C07281=1053.248,31.151,424.768,170.927,31.729,155.954
C07282=1053.242,30.901,424.785,170.926,31.727,155.954
C07283=1053.236,30.652,424.801,170.924,31.725,155.953
C07284=1053.230,30.403,424.817,170.922,31.723,155.953
C07285=1053.224,30.153,424.833,170.920,31.720,155.953
C07286=1053.217,29.868,424.851,170.919,31.718,155.952
C07287=1053.209,29.582,424.870,170.917,31.716,155.952
C07288=1053.203,29.296,424.888,170.915,31.714,155.952
C07289=1053.196,29.011,424.906,170.914,31.711,155.951
C07290=1053.189,28.761,424.923,170.912,31.709,155.951
C07291=1053.184,28.511,424.938,170.910,31.707,155.951
C07292=1053.177,28.262,424.954,170.909,31.704,155.950
C07293=1053.171,28.012,424.970,170.907,31.702,155.950
C07294=1053.165,27.763,424.987,170.905,31.700,155.950
C07295=1053.158,27.514,425.002,170.903,31.698,155.949
C07296=1053.153,27.264,425.018,170.902,31.696,155.949
C07297=1053.146,27.015,425.034,170.900,31.694,155.949
C07298=1053.140,26.765,425.050,170.899,31.692,155.949
C07299=1053.134,26.516,425.066,170.897,31.690,155.948
C07300=1053.127,26.267,425.082,170.896,31.688,155.948
C07301=1053.122,26.017,425.097,170.894,31.686,155.948
C07302=1053.114,25.767,425.113,170.892,31.684,155.947
C07303=1053.108,25.518,425.130,170.891,31.682,155.947
C07304=1053.103,25.269,425.146,170.889,31.679,155.947
C07305=1053.096,25.019,425.161,170.887,31.677,155.946
C07306=1053.090,24.770,425.177,170.885,31.675,155.946
C07307=1053.084,24.521,425.193,170.884,31.673,155.946
C07308=1053.078,24.271,425.208,170.883,31.671,155.945
C07309=1053.071,24.022,425.224,170.881,31.669,155.945
C07310=1053.065,23.772,425.240,170.880,31.667,155.945
C07311=1053.059,23.523,425.256,170.878,31.665,155.945
C07312=1053.053,23.273,425.271,170.876,31.663,155.944
C07313=1053.047,23.024,425.288,170.874,31.660,155.944
C07314=1053.040,22.775,425.303,170.873,31.659,155.944
C07315=1053.035,22.525,425.319,170.871,31.656,155.943
C07316=1053.028,22.276,425.334,170.869,31.654,155.943
C07317=1053.022,22.026,425.350,170.868,31.652,155.943
C07318=1053.016,21.777,425.366,170.867,31.650,155.942
C07319=1053.010,21.528,425.382,170.865,31.648,155.942
C07320=1053.003,21.278,425.397,170.863,31.645,155.942
C07321=1052.997,21.029,425.413,170.862,31.644,155.942
C07322=1052.991,20.779,425.429,170.860,31.641,155.941
C07323=1052.985,20.530,425.444,170.858,31.639,155.941
C07324=1052.979,20.280,425.461,170.856,31.637,155.941
C07325=1052.973,20.030,425.475,170.855,31.635,155.940
C07326=1052.967,19.781,425.492,170.853,31.633,155.940
C07327=1052.960,19.531,425.507,170.852,31.631,155.940
C07328=1052.954,19.282,425.522,170.850,31.629,155.939
C07329=1052.948,19.032,425.538,170.849,31.627,155.939
C07330=1052.941,18.783,425.554,170.847,31.625,155.939
C07331=1052.936,18.533,425.569,170.845,31.623,155.939
C07332=1052.929,18.284,425.585,170.843,31.621,155.938
C07333=1052.923,18.035,425.600,170.842,31.619,155.938
C07334=1052.917,17.785,425.616,170.840,31.617,155.938
C07335=1052.910,17.536,425.631,170.838,31.615,155.937
C07336=1052.905,17.287,425.647,170.837,31.613,155.937
C07337=1052.898,17.037,425.662,170.836,31.611,155.937
C07338=1052.892,16.788,425.677,170.834,31.608,155.936
C07339=1052.886,16.538,425.693,170.832,31.606,155.936
C07340=1052.879,16.289,425.709,170.830,31.604,155.936
C07341=1052.874,16.039,425.724,170.829,31.602,155.936
C07342=1052.867,15.790,425.740,170.827,31.600,155.935
C07343=1052.861,15.541,425.755,170.825,31.598,155.935
C07344=1052.855,15.291,425.770,170.823,31.596,155.935
C07345=1052.848,15.042,425.786,170.823,31.594,155.934
C07346=1052.842,14.792,425.801,170.821,31.592,155.934
C07347=1052.836,14.543,425.817,170.819,31.590,155.934
C07348=1052.830,14.294,425.832,170.817,31.588,155.934
C07349=1052.824,14.044,425.847,170.816,31.586,155.933
C07350=1052.816,13.760,425.865,170.814,31.584,155.933
C07351=1052.809,13.475,425.882,170.812,31.581,155.933
C07352=1052.802,13.191,425.900,170.810,31.579,155.932
C07353=1052.795,12.906,425.917,170.808,31.577,155.932
C07354=1052.789,12.656,425.932,170.807,31.575,155.932
C07355=1052.782,12.407,425.948,170.805,31.573,155.931
C07356=1052.776,12.158,425.963,170.803,31.571,155.931
C07357=1052.769,11.908,425.978,170.802,31.569,155.931
C07358=1052.764,11.658,425.993,170.800,31.566,155.931
C07359=1052.757,11.409,426.009,170.798,31.564,155.930
C07360=1052.751,11.160,426.023,170.796,31.563,155.930
C07361=1052.745,10.910,426.038,170.794,31.561,155.930
C07362=1052.738,10.661,426.054,170.793,31.559,155.929
C07363=1052.732,10.412,426.069,170.792,31.557,155.929
C07364=1052.725,10.162,426.084,170.790,31.555,155.929
C07365=1052.719,9.912,426.099,170.788,31.553,155.929
C07366=1052.713,9.662,426.114,170.787,31.551,155.928
C07367=1052.707,9.414,426.130,170.785,31.548,155.928
C07368=1052.701,9.164,426.145,170.783,31.547,155.928
C07369=1052.695,8.915,426.159,170.781,31.545,155.928
C07370=1052.688,8.665,426.174,170.779,31.543,155.927
C07371=1052.682,8.415,426.189,170.778,31.541,155.927
C07372=1052.675,8.166,426.205,170.777,31.539,155.927
C07373=1052.669,7.917,426.220,170.775,31.537,155.926
C07374=1052.664,7.668,426.235,170.773,31.534,155.926
C07375=1052.657,7.418,426.250,170.772,31.533,155.926
C07376=1052.651,7.168,426.265,170.770,31.531,155.926
C07377=1052.645,6.919,426.280,170.768,31.529,155.925
C07378=1052.638,6.669,426.295,170.766,31.527,155.925
C07379=1052.632,6.421,426.310,170.764,31.525,155.925
C07380=1052.626,6.171,426.325,170.763,31.523,155.924
C07381=1052.619,5.921,426.340,170.762,31.521,155.924
C07382=1052.613,5.672,426.355,170.760,31.519,155.924
C07383=1052.607,5.422,426.370,170.758,31.516,155.924
C07384=1052.602,5.173,426.385,170.757,31.515,155.923
C07385=1052.595,4.923,426.400,170.755,31.513,155.923
C07386=1052.589,4.673,426.415,170.753,31.511,155.923
C07387=1052.582,4.424,426.430,170.751,31.509,155.922
C07388=1052.577,4.175,426.445,170.749,31.507,155.922
C07389=1052.570,3.925,426.460,170.749,31.505,155.922
C07390=1052.564,3.675,426.475,170.747,31.503,155.922
C07391=1052.557,3.426,426.489,170.745,31.500,155.921
C07392=1052.552,3.177,426.504,170.743,31.499,155.921
C07393=1052.545,2.927,426.519,170.741,31.497,155.921
C07394=1052.539,2.678,426.534,170.740,31.495,155.921
C07395=1052.533,2.429,426.549,170.738,31.493,155.920
C07396=1052.527,2.179,426.563,170.736,31.491,155.920
C07397=1052.521,1.929,426.579,170.734,31.489,155.920
C07398=1052.515,1.679,426.594,170.733,31.487,155.919
C07399=1052.509,1.430,426.609,170.732,31.485,155.919
C07400=1052.503,1.181,426.623,170.730,31.483,155.919
C07401=1052.496,0.931,426.638,170.728,31.481,155.919
C07402=1052.490,0.682,426.653,170.726,31.479,155.918
C07403=1052.484,0.432,426.668,170.725,31.477,155.918
C07404=1052.478,0.183,426.683,170.723,31.475,155.918
C07405=1052.472,-0.066,426.697,170.721,31.473,155.917
C07406=1052.465,-0.316,426.712,170.719,31.471,155.917
C07407=1052.459,-0.566,426.727,170.718,31.469,155.917
C07408=1052.453,-0.814,426.742,170.717,31.467,155.917
C07409=1052.447,-1.065,426.756,170.715,31.465,155.916
C07410=1052.441,-1.314,426.771,170.713,31.463,155.916
C07411=1052.435,-1.563,426.786,170.711,31.461,155.916
C07412=1052.429,-1.813,426.801,170.709,31.459,155.916
C07413=1052.422,-2.063,426.816,170.708,31.457,155.915
C07414=1052.415,-2.345,426.832,170.705,31.454,155.915
C07415=1052.409,-2.628,426.848,170.704,31.452,155.915
C07416=1052.402,-2.910,426.865,170.702,31.450,155.914
C07417=1052.395,-3.193,426.882,170.700,31.447,155.914
C07418=1052.389,-3.442,426.897,170.699,31.446,155.914
C07419=1052.383,-3.692,426.911,170.697,31.444,155.914
C07420=1052.377,-3.941,426.926,170.695,31.442,155.913
C07421=1052.369,-4.191,426.940,170.693,31.440,155.913
C07422=1052.364,-4.440,426.955,170.691,31.438,155.913
C07423=1052.358,-4.690,426.969,170.690,31.436,155.912
C07424=1052.351,-4.940,426.984,170.689,31.435,155.912
C07425=1052.345,-5.188,426.998,170.687,31.433,155.912
C07426=1052.338,-5.438,427.013,170.685,31.431,155.912
C07427=1052.333,-5.688,427.027,170.683,31.429,155.912
C07428=1052.326,-5.937,427.042,170.681,31.427,155.911
C07429=1052.319,-6.187,427.056,170.679,31.425,155.911
C07430=1052.314,-6.436,427.070,170.678,31.423,155.911
C07431=1052.307,-6.686,427.085,170.676,31.421,155.911
C07432=1052.301,-6.935,427.100,170.675,31.419,155.910
C07433=1052.295,-7.185,427.113,170.673,31.417,155.910
C07434=1052.288,-7.434,427.128,170.671,31.416,155.910
C07435=1052.283,-7.683,427.143,170.669,31.414,155.909
C07436=1052.276,-7.933,427.156,170.667,31.411,155.909
C07437=1052.270,-8.183,427.171,170.666,31.410,155.909
C07438=1052.264,-8.432,427.186,170.664,31.408,155.909
C07439=1052.258,-8.682,427.200,170.662,31.406,155.908
C07440=1052.251,-8.931,427.214,170.660,31.404,155.908
C07441=1052.245,-9.181,427.228,170.659,31.402,155.908
C07442=1052.239,-9.431,427.243,170.657,31.400,155.908
C07443=1052.232,-9.679,427.257,170.656,31.399,155.907
C07444=1052.226,-9.930,427.271,170.654,31.397,155.907
C07445=1052.220,-10.179,427.286,170.652,31.395,155.907
C07446=1052.213,-10.429,427.300,170.650,31.393,155.907
C07447=1052.208,-10.678,427.314,170.648,31.391,155.906
C07448=1052.202,-10.928,427.328,170.646,31.389,155.906
C07449=1052.195,-11.176,427.342,170.645,31.387,155.906
C07450=1052.189,-11.427,427.357,170.644,31.385,155.906
C07451=1052.183,-11.676,427.371,170.642,31.384,155.906
C07452=1052.177,-11.926,427.385,170.640,31.382,155.905
C07453=1052.171,-12.175,427.399,170.638,31.380,155.905
C07454=1052.165,-12.425,427.414,170.636,31.378,155.905
C07455=1052.159,-12.674,427.428,170.634,31.376,155.905
C07456=1052.152,-12.924,427.442,170.633,31.374,155.904
C07457=1052.146,-13.173,427.456,170.631,31.372,155.904
C07458=1052.140,-13.423,427.471,170.630,31.370,155.904
C07459=1052.134,-13.672,427.485,170.628,31.368,155.903
C07460=1052.127,-13.922,427.499,170.626,31.367,155.903
C07461=1052.122,-14.171,427.513,170.624,31.365,155.903
C07462=1052.115,-14.421,427.527,170.622,31.362,155.903
C07463=1052.109,-14.670,427.542,170.621,31.361,155.903
C07464=1052.102,-14.920,427.555,170.619,31.359,155.902
C07465=1052.097,-15.169,427.569,170.617,31.358,155.902
C07466=1052.090,-15.419,427.584,170.616,31.355,155.902
C07467=1052.084,-15.668,427.597,170.614,31.354,155.902
C07468=1052.077,-15.918,427.612,170.612,31.352,155.901
C07469=1052.072,-16.167,427.626,170.610,31.350,155.901
C07470=1052.065,-16.417,427.639,170.608,31.348,155.901
C07471=1052.059,-16.666,427.654,170.606,31.347,155.901
C07472=1052.052,-16.916,427.667,170.605,31.345,155.900
C07473=1052.047,-17.166,427.681,170.603,31.343,155.900
C07474=1052.040,-17.415,427.696,170.602,31.341,155.900
C07475=1052.034,-17.665,427.709,170.600,31.340,155.900
C07476=1052.027,-17.915,427.723,170.598,31.337,155.900
C07477=1052.021,-18.164,427.736,170.596,31.336,155.899
C07478=1052.014,-18.445,427.752,170.594,31.334,155.899
C07479=1052.007,-18.725,427.769,170.592,31.332,155.899
C07480=1052.000,-19.007,427.784,170.590,31.330,155.898
C07481=1051.993,-19.288,427.800,170.588,31.327,155.898
C07482=1051.987,-19.537,427.813,170.586,31.326,155.898
C07483=1051.980,-19.787,427.827,170.585,31.324,155.898
C07484=1051.975,-20.036,427.841,170.583,31.322,155.898
C07485=1051.967,-20.286,427.855,170.581,31.320,155.897
C07486=1051.962,-20.535,427.869,170.579,31.319,155.897
C07487=1051.956,-20.785,427.882,170.577,31.317,155.897
C07488=1051.949,-21.035,427.896,170.575,31.315,155.897
C07489=1051.943,-21.284,427.910,170.574,31.314,155.896
C07490=1051.936,-21.534,427.924,170.572,31.312,155.896
C07491=1051.931,-21.783,427.938,170.571,31.310,155.896
C07492=1051.925,-22.032,427.951,170.569,31.308,155.896
C07493=1051.918,-22.282,427.965,170.567,31.306,155.896
C07494=1051.912,-22.532,427.979,170.565,31.304,155.895
C07495=1051.906,-22.781,427.992,170.563,31.303,155.895
C07496=1051.900,-23.031,428.007,170.561,31.301,155.895
C07497=1051.894,-23.280,428.020,170.559,31.299,155.895
C07498=1051.887,-23.529,428.034,170.557,31.297,155.894
C07499=1051.881,-23.780,428.048,170.557,31.296,155.894
C07500=1051.875,-24.029,428.061,170.555,31.293,155.894
C07501=1051.869,-24.278,428.074,170.553,31.292,155.894
C07502=1051.863,-24.528,428.089,170.551,31.290,155.894
C07503=1051.857,-24.778,428.102,170.549,31.288,155.893
C07504=1051.850,-25.027,428.115,170.547,31.287,155.893
C07505=1051.844,-25.277,428.129,170.545,31.285,155.893
C07506=1051.838,-25.526,428.143,170.543,31.283,155.893
C07507=1051.832,-25.775,428.157,170.542,31.281,155.892
C07508=1051.825,-26.025,428.171,170.540,31.280,155.892
C07509=1051.819,-26.275,428.184,170.538,31.277,155.892
C07510=1051.814,-26.524,428.198,170.537,31.276,155.892
C07511=1051.807,-26.774,428.212,170.535,31.275,155.892
C07512=1051.801,-27.024,428.225,170.533,31.272,155.891
C07513=1051.795,-27.273,428.238,170.531,31.271,155.891
C07514=1051.788,-27.523,428.252,170.529,31.269,155.891
C07515=1051.782,-27.772,428.266,170.527,31.267,155.891
C07516=1051.776,-28.022,428.279,170.526,31.266,155.891
C07517=1051.769,-28.272,428.293,170.524,31.264,155.890
C07518=1051.763,-28.521,428.305,170.522,31.262,155.890
C07519=1051.757,-28.771,428.318,170.520,31.261,155.890
C07520=1051.751,-29.020,428.332,170.518,31.259,155.890
C07521=1051.744,-29.270,428.345,170.516,31.258,155.890
C07522=1051.739,-29.520,428.359,170.514,31.255,155.889
C07523=1051.732,-29.769,428.372,170.512,31.254,155.889
C07524=1051.726,-30.019,428.386,170.511,31.252,155.889
C07525=1051.719,-30.268,428.399,170.510,31.250,155.889
C07526=1051.713,-30.517,428.413,170.508,31.249,155.888
C07527=1051.707,-30.767,428.426,170.506,31.247,155.888
C07528=1051.700,-31.017,428.439,170.504,31.246,155.888
C07529=1051.694,-31.266,428.452,170.502,31.244,155.888
C07530=1051.688,-31.516,428.465,170.500,31.242,155.888
C07531=1051.682,-31.765,428.479,170.498,31.241,155.888
C07532=1051.676,-32.015,428.493,170.496,31.239,155.887
C07533=1051.669,-32.264,428.506,170.495,31.237,155.887
C07534=1051.664,-32.514,428.519,170.493,31.236,155.887
C07535=1051.657,-32.764,428.532,170.491,31.234,155.887
C07536=1051.651,-33.014,428.546,170.489,31.232,155.887
C07537=1051.644,-33.263,428.559,170.487,31.230,155.886
C07538=1051.638,-33.512,428.572,170.485,31.229,155.886
C07539=1051.632,-33.762,428.585,170.483,31.227,155.886
C07540=1051.626,-34.011,428.598,170.481,31.226,155.886
C07541=1051.619,-34.261,428.612,170.480,31.224,155.886
C07542=1051.613,-34.542,428.627,170.478,31.222,155.885
C07543=1051.606,-34.822,428.642,170.476,31.220,155.885
C07544=1051.599,-35.102,428.656,170.474,31.218,155.885
C07545=1051.592,-35.382,428.671,170.472,31.216,155.885
C07546=1051.586,-35.632,428.684,170.470,31.215,155.884
C07547=1051.580,-35.881,428.697,170.468,31.213,155.884
C07548=1051.573,-36.130,428.710,170.466,31.212,155.884
C07549=1051.567,-36.380,428.723,170.465,31.210,155.884
C07550=1051.561,-36.630,428.737,170.463,31.208,155.884
C07551=1051.554,-36.879,428.750,170.461,31.207,155.884
C07552=1051.548,-37.129,428.762,170.459,31.205,155.883
C07553=1051.542,-37.379,428.776,170.457,31.203,155.883
C07554=1051.537,-37.628,428.789,170.455,31.201,155.883
C07555=1051.531,-37.878,428.802,170.453,31.200,155.883
C07556=1051.525,-38.127,428.815,170.451,31.198,155.883
C07557=1051.518,-38.376,428.829,170.449,31.197,155.882
C07558=1051.512,-38.627,428.841,170.448,31.195,155.882
C07559=1051.506,-38.876,428.855,170.446,31.193,155.882
C07560=1051.499,-39.126,428.867,170.444,31.192,155.882
C07561=1051.493,-39.375,428.880,170.442,31.190,155.882
C07562=1051.487,-39.624,428.893,170.440,31.189,155.881
C07563=1051.481,-39.874,428.906,170.438,31.187,155.881
C07564=1051.475,-40.124,428.919,170.436,31.186,155.881
C07565=1051.468,-40.374,428.932,170.434,31.184,155.881
C07566=1051.461,-40.623,428.945,170.433,31.183,155.881
C07567=1051.455,-40.873,428.957,170.431,31.181,155.881
C07568=1051.449,-41.122,428.970,170.429,31.180,155.880
C07569=1051.443,-41.372,428.983,170.427,31.178,155.880
C07570=1051.437,-41.621,428.996,170.425,31.177,155.880
C07571=1051.430,-41.871,429.008,170.423,31.175,155.880
C07572=1051.424,-42.120,429.022,170.421,31.173,155.880
C07573=1051.418,-42.370,429.034,170.419,31.171,155.880
C07574=1051.411,-42.620,429.048,170.417,31.170,155.879
C07575=1051.405,-42.870,429.060,170.416,31.168,155.879
C07576=1051.399,-43.119,429.074,170.414,31.167,155.879
C07577=1051.392,-43.369,429.086,170.412,31.165,155.879
C07578=1051.386,-43.618,429.099,170.410,31.164,155.879
C07579=1051.380,-43.868,429.111,170.408,31.162,155.879
C07580=1051.374,-44.118,429.124,170.406,31.161,155.878
C07581=1051.367,-44.367,429.137,170.404,31.159,155.878
C07582=1051.362,-44.617,429.149,170.402,31.158,155.878
C07583=1051.355,-44.866,429.162,170.401,31.156,155.878
C07584=1051.349,-45.116,429.175,170.399,31.155,155.878
C07585=1051.344,-45.366,429.187,170.397,31.153,155.878
C07586=1051.337,-45.615,429.200,170.395,31.152,155.877
C07587=1051.331,-45.865,429.213,170.393,31.150,155.877
C07588=1051.324,-46.114,429.226,170.391,31.148,155.877
C07589=1051.319,-46.364,429.239,170.389,31.147,155.877
C07590=1051.312,-46.613,429.251,170.387,31.145,155.877
C07591=1051.306,-46.863,429.264,170.385,31.144,155.877
C07592=1051.300,-47.112,429.276,170.384,31.142,155.876
C07593=1051.294,-47.362,429.289,170.382,31.141,155.876
C07594=1051.288,-47.612,429.302,170.380,31.139,155.876
C07595=1051.281,-47.861,429.314,170.378,31.138,155.876
C07596=1051.275,-48.111,429.327,170.376,31.136,155.876
C07597=1051.269,-48.361,429.339,170.374,31.135,155.876
C07598=1051.263,-48.610,429.352,170.372,31.133,155.875
C07599=1051.256,-48.860,429.364,170.370,31.132,155.875
C07600=1051.250,-49.110,429.377,170.369,31.130,155.875
C07601=1051.245,-49.360,429.390,170.367,31.129,155.875
C07602=1051.238,-49.609,429.403,170.365,31.127,155.875
C07603=1051.232,-49.858,429.415,170.363,31.126,155.875
C07604=1051.226,-50.108,429.427,170.361,31.125,155.875
C07605=1051.220,-50.358,429.440,170.359,31.123,155.874
C07606=1051.212,-50.639,429.453,170.357,31.122,155.874
C07607=1051.205,-50.919,429.468,170.354,31.120,155.874
C07608=1051.198,-51.199,429.482,170.352,31.118,155.874
C07609=1051.191,-51.480,429.496,170.351,31.117,155.874
C07610=1051.184,-51.729,429.508,170.349,31.115,155.874
C07611=1051.178,-51.979,429.520,170.347,31.114,155.873
C07612=1051.172,-52.229,429.532,170.345,31.112,155.873
C07613=1051.166,-52.479,429.545,170.343,31.111,155.873
C07614=1051.159,-52.728,429.557,170.341,31.110,155.873
C07615=1051.153,-52.978,429.569,170.339,31.108,155.873
C07616=1051.147,-53.228,429.581,170.337,31.107,155.873
C07617=1051.140,-53.477,429.594,170.334,31.106,155.873
C07618=1051.134,-53.726,429.606,170.333,31.104,155.872
C07619=1051.127,-53.976,429.618,170.331,31.103,155.872
C07620=1051.121,-54.226,429.631,170.329,31.102,155.872
C07621=1051.115,-54.476,429.643,170.327,31.100,155.872
C07622=1051.108,-54.725,429.655,170.325,31.099,155.872
C07623=1051.103,-54.974,429.667,170.323,31.098,155.872
C07624=1051.096,-55.224,429.679,170.321,31.096,155.872
C07625=1051.090,-55.474,429.692,170.319,31.095,155.872
C07626=1051.083,-55.723,429.703,170.317,31.094,155.872
C07627=1051.077,-55.973,429.715,170.316,31.092,155.871
C07628=1051.071,-56.223,429.728,170.314,31.091,155.871
C07629=1051.064,-56.472,429.740,170.312,31.089,155.871
C07630=1051.058,-56.722,429.753,170.310,31.088,155.871
C07631=1051.052,-56.972,429.764,170.308,31.087,155.871
C07632=1051.045,-57.221,429.776,170.306,31.085,155.871
C07633=1051.040,-57.471,429.789,170.304,31.084,155.871
C07634=1051.033,-57.720,429.801,170.301,31.083,155.870
C07635=1051.026,-57.970,429.813,170.300,31.081,155.870
C07636=1051.021,-58.220,429.825,170.298,31.080,155.870
C07637=1051.014,-58.469,429.837,170.296,31.079,155.870
C07638=1051.008,-58.719,429.850,170.294,31.078,155.870
C07639=1051.002,-58.969,429.861,170.292,31.076,155.870
C07640=1050.996,-59.218,429.872,170.290,31.075,155.870
C07641=1050.990,-59.468,429.885,170.288,31.074,155.870
C07642=1050.983,-59.718,429.897,170.286,31.072,155.869
C07643=1050.976,-59.967,429.909,170.284,31.071,155.869
C07644=1050.971,-60.217,429.921,170.282,31.070,155.869
C07645=1050.964,-60.467,429.933,170.281,31.068,155.869
C07646=1050.958,-60.715,429.945,170.279,31.067,155.869
C07647=1050.952,-60.966,429.957,170.277,31.066,155.869
C07648=1050.946,-61.215,429.969,170.275,31.064,155.869
C07649=1050.939,-61.465,429.981,170.272,31.063,155.869
C07650=1050.934,-61.714,429.993,170.270,31.062,155.869
C07651=1050.927,-61.964,430.005,170.268,31.060,155.868
C07652=1050.920,-62.213,430.017,170.266,31.059,155.868
C07653=1050.915,-62.464,430.029,170.264,31.058,155.868
C07654=1050.908,-62.713,430.041,170.263,31.057,155.868
C07655=1050.902,-62.962,430.052,170.261,31.055,155.868
C07656=1050.896,-63.212,430.065,170.259,31.054,155.868
C07657=1050.890,-63.462,430.076,170.257,31.053,155.868
C07658=1050.883,-63.712,430.088,170.255,31.051,155.868
C07659=1050.878,-63.961,430.100,170.253,31.050,155.868
C07660=1050.871,-64.211,430.112,170.251,31.049,155.867
C07661=1050.865,-64.461,430.123,170.248,31.048,155.867
C07662=1050.860,-64.710,430.136,170.246,31.046,155.867
C07663=1050.853,-64.960,430.148,170.245,31.045,155.867
C07664=1050.846,-65.209,430.160,170.243,31.044,155.867
C07665=1050.840,-65.459,430.171,170.241,31.042,155.867
C07666=1050.835,-65.709,430.183,170.239,31.041,155.867
C07667=1050.828,-65.958,430.195,170.237,31.040,155.867
C07668=1050.822,-66.208,430.206,170.235,31.039,155.867
C07669=1050.816,-66.458,430.218,170.233,31.037,155.866
C07670=1050.809,-66.739,430.231,170.230,31.036,155.866
C07671=1050.801,-67.021,430.245,170.228,31.035,155.866
C07672=1050.795,-67.303,430.258,170.227,31.033,155.866
C07673=1050.788,-67.585,430.272,170.224,31.032,155.866
C07674=1050.782,-67.835,430.283,170.222,31.031,155.866
C07675=1050.776,-68.084,430.294,170.220,31.029,155.866
C07676=1050.770,-68.334,430.307,170.218,31.028,155.866
C07677=1050.764,-68.585,430.318,170.216,31.027,155.865
C07678=1050.758,-68.833,430.330,170.214,31.026,155.865
C07679=1050.751,-69.083,430.342,170.212,31.024,155.865
C07680=1050.745,-69.333,430.354,170.210,31.023,155.865
C07681=1050.739,-69.582,430.365,170.209,31.022,155.865
C07682=1050.733,-69.833,430.376,170.207,31.021,155.865
C07683=1050.727,-70.081,430.388,170.204,31.019,155.865
C07684=1050.721,-70.332,430.400,170.202,31.018,155.865
C07685=1050.715,-70.581,430.412,170.200,31.017,155.865
C07686=1050.709,-70.831,430.423,170.198,31.016,155.865
C07687=1050.702,-71.081,430.435,170.196,31.014,155.864
C07688=1050.697,-71.330,430.447,170.194,31.013,155.864
C07689=1050.691,-71.580,430.458,170.192,31.012,155.864
C07690=1050.685,-71.829,430.470,170.191,31.011,155.864
C07691=1050.678,-72.079,430.481,170.189,31.009,155.864
C07692=1050.673,-72.329,430.493,170.187,31.008,155.864
C07693=1050.667,-72.578,430.504,170.184,31.007,155.864
C07694=1050.660,-72.829,430.516,170.182,31.006,155.864
C07695=1050.654,-73.077,430.527,170.180,31.005,155.864
C07696=1050.648,-73.328,430.538,170.178,31.003,155.864
C07697=1050.643,-73.577,430.551,170.176,31.002,155.864
C07698=1050.636,-73.827,430.562,170.174,31.001,155.863
C07699=1050.630,-74.076,430.573,170.173,31.000,155.863
C07700=1050.624,-74.326,430.585,170.171,30.999,155.863
C07701=1050.618,-74.576,430.596,170.169,30.998,155.863
C07702=1050.611,-74.825,430.607,170.166,30.996,155.863
C07703=1050.605,-75.075,430.619,170.164,30.995,155.863
C07704=1050.599,-75.325,430.630,170.162,30.995,155.863
C07705=1050.593,-75.574,430.642,170.160,30.994,155.863
C07706=1050.587,-75.824,430.652,170.158,30.992,155.863
C07707=1050.580,-76.073,430.664,170.156,30.991,155.863
C07708=1050.574,-76.324,430.676,170.154,30.990,155.863
C07709=1050.568,-76.573,430.687,170.152,30.989,155.863
C07710=1050.562,-76.823,430.698,170.150,30.988,155.862
C07711=1050.556,-77.072,430.709,170.148,30.987,155.862
C07712=1050.550,-77.322,430.721,170.146,30.986,155.862
C07713=1050.544,-77.572,430.731,170.144,30.985,155.862
C07714=1050.537,-77.821,430.743,170.142,30.983,155.862
C07715=1050.531,-78.071,430.754,170.140,30.982,155.862
C07716=1050.525,-78.321,430.766,170.138,30.981,155.862
C07717=1050.519,-78.571,430.776,170.135,30.980,155.862
C07718=1050.513,-78.820,430.788,170.133,30.979,155.862
C07719=1050.506,-79.069,430.799,170.132,30.978,155.862
C07720=1050.500,-79.319,430.810,170.130,30.977,155.862
C07721=1050.494,-79.569,430.821,170.128,30.976,155.862
C07722=1050.487,-79.819,430.833,170.126,30.975,155.862
C07723=1050.482,-80.068,430.844,170.124,30.974,155.862
C07724=1050.475,-80.318,430.855,170.121,30.973,155.862
C07725=1050.470,-80.568,430.866,170.119,30.972,155.862
C07726=1050.463,-80.818,430.876,170.117,30.971,155.862
C07727=1050.457,-81.067,430.887,170.115,30.970,155.861
C07728=1050.450,-81.317,430.899,170.113,30.969,155.861
C07729=1050.444,-81.566,430.910,170.112,30.969,155.861
C07730=1050.437,-81.816,430.921,170.109,30.967,155.861
C07731=1050.432,-82.066,430.932,170.107,30.967,155.861
C07732=1050.425,-82.316,430.943,170.105,30.966,155.861
C07733=1050.419,-82.565,430.953,170.103,30.965,155.861
C07734=1050.412,-82.849,430.966,170.100,30.964,155.861
C07735=1050.405,-83.133,430.978,170.098,30.963,155.861
C07736=1050.398,-83.417,430.991,170.096,30.961,155.861
C07737=1050.391,-83.702,431.003,170.093,30.960,155.861
C07738=1050.384,-83.951,431.014,170.091,30.959,155.861
C07739=1050.378,-84.200,431.025,170.090,30.958,155.861
C07740=1050.372,-84.451,431.037,170.088,30.957,155.861
C07741=1050.366,-84.700,431.047,170.085,30.956,155.861
C07742=1050.359,-84.950,431.058,170.083,30.955,155.861
C07743=1050.353,-85.199,431.069,170.081,30.955,155.861
C07744=1050.347,-85.449,431.080,170.079,30.954,155.861
C07745=1050.340,-85.699,431.090,170.077,30.953,155.861
C07746=1050.334,-85.948,431.101,170.075,30.952,155.861
C07747=1050.328,-86.198,431.113,170.072,30.951,155.861
C07748=1050.322,-86.448,431.123,170.070,30.950,155.861
C07749=1050.316,-86.697,431.134,170.069,30.949,155.861
C07750=1050.310,-86.947,431.145,170.067,30.948,155.860
C07751=1050.303,-87.197,431.155,170.065,30.947,155.860
C07752=1050.297,-87.447,431.166,170.063,30.947,155.860
C07753=1050.291,-87.697,431.177,170.060,30.945,155.860
C07754=1050.285,-87.946,431.187,170.058,30.945,155.860
C07755=1050.278,-88.196,431.198,170.056,30.944,155.860
C07756=1050.273,-88.446,431.209,170.054,30.943,155.860
C07757=1050.266,-88.695,431.219,170.052,30.942,155.860
C07758=1050.260,-88.945,431.231,170.050,30.941,155.860
C07759=1050.254,-89.194,431.241,170.047,30.940,155.860
C07760=1050.248,-89.444,431.252,170.046,30.939,155.860
C07761=1050.241,-89.694,431.263,170.044,30.939,155.860
C07762=1050.236,-89.944,431.273,170.042,30.938,155.860
C07763=1050.229,-90.193,431.283,170.040,30.937,155.860
C07764=1050.223,-90.443,431.295,170.037,30.936,155.860
C07765=1050.217,-90.693,431.306,170.035,30.935,155.860
C07766=1050.211,-90.942,431.316,170.033,30.934,155.860
C07767=1050.205,-91.192,431.327,170.031,30.933,155.860
C07768=1050.198,-91.442,431.337,170.029,30.933,155.860
C07769=1050.193,-91.691,431.348,170.027,30.932,155.860
C07770=1050.187,-91.941,431.358,170.024,30.931,155.860
C07771=1050.180,-92.191,431.369,170.023,30.930,155.860
C07772=1050.174,-92.440,431.380,170.021,30.929,155.860
C07773=1050.169,-92.690,431.390,170.019,30.928,155.860
C07774=1050.162,-92.940,431.400,170.017,30.927,155.860
C07775=1050.156,-93.190,431.412,170.014,30.927,155.860
C07776=1050.149,-93.439,431.422,170.012,30.926,155.860
C07777=1050.144,-93.689,431.432,170.010,30.925,155.860
C07778=1050.138,-93.939,431.443,170.008,30.924,155.860
C07779=1050.131,-94.188,431.454,170.006,30.923,155.860
C07780=1050.125,-94.438,431.464,170.004,30.923,155.860
C07781=1050.119,-94.688,431.474,170.001,30.922,155.860
C07782=1050.113,-94.937,431.485,170.000,30.921,155.860
C07783=1050.107,-95.187,431.496,169.998,30.920,155.860
C07784=1050.101,-95.437,431.506,169.996,30.920,155.860
C07785=1050.095,-95.687,431.517,169.994,30.919,155.860
C07786=1050.089,-95.936,431.527,169.991,30.918,155.860
C07787=1050.083,-96.186,431.537,169.989,30.917,155.860
C07788=1050.077,-96.436,431.548,169.987,30.917,155.860
C07789=1050.070,-96.685,431.559,169.985,30.916,155.860
C07790=1050.065,-96.936,431.569,169.983,30.915,155.860
C07791=1050.059,-97.185,431.579,169.981,30.914,155.860
C07792=1050.053,-97.434,431.590,169.978,30.913,155.860
C07793=1050.047,-97.684,431.599,169.977,30.912,155.860
C07794=1050.040,-97.934,431.611,169.975,30.911,155.860
C07795=1050.034,-98.184,431.620,169.973,30.911,155.860
C07796=1050.028,-98.433,431.631,169.970,30.910,155.860
C07797=1050.022,-98.683,431.641,169.968,30.910,155.860
C07798=1050.015,-98.970,431.653,169.966,30.909,155.860
C07799=1050.008,-99.256,431.664,169.963,30.908,155.860
C07800=1050.001,-99.542,431.676,169.961,30.907,155.860
C07801=1049.993,-99.829,431.688,169.958,30.906,155.860
C07802=1049.987,-100.078,431.699,169.956,30.906,155.860
C07803=1049.981,-100.328,431.708,169.954,30.905,155.860
C07804=1049.975,-100.577,431.719,169.952,30.905,155.860
C07805=1049.969,-100.828,431.729,169.950,30.904,155.860
C07806=1049.962,-101.077,431.739,169.948,30.903,155.860
C07807=1049.956,-101.327,431.749,169.946,30.902,155.860
C07808=1049.950,-101.577,431.759,169.944,30.902,155.860
C07809=1049.944,-101.826,431.769,169.941,30.901,155.860
C07810=1049.938,-102.076,431.779,169.939,30.901,155.860
C07811=1049.932,-102.325,431.790,169.937,30.900,155.860
C07812=1049.926,-102.575,431.799,169.935,30.900,155.860
C07813=1049.919,-102.825,431.810,169.933,30.899,155.860
C07814=1049.913,-103.075,431.820,169.930,30.898,155.860
C07815=1049.907,-103.324,431.830,169.928,30.897,155.860
C07816=1049.901,-103.574,431.840,169.926,30.897,155.860
C07817=1049.895,-103.824,431.850,169.925,30.896,155.860
C07818=1049.889,-104.073,431.860,169.922,30.896,155.860
C07819=1049.883,-104.323,431.870,169.920,30.895,155.860
C07820=1049.876,-104.573,431.880,169.918,30.894,155.860
C07821=1049.871,-104.823,431.890,169.916,30.894,155.860
C07822=1049.865,-105.072,431.900,169.914,30.893,155.860
C07823=1049.857,-105.322,431.911,169.911,30.893,155.860
C07824=1049.851,-105.572,431.920,169.909,30.892,155.860
C07825=1049.846,-105.822,431.930,169.907,30.891,155.860
C07826=1049.840,-106.072,431.940,169.905,30.891,155.860
C07827=1049.833,-106.321,431.950,169.903,30.890,155.860
C07828=1049.827,-106.571,431.960,169.900,30.890,155.860
C07829=1049.822,-106.821,431.970,169.898,30.889,155.860
C07830=1049.815,-107.070,431.980,169.897,30.888,155.860
C07831=1049.809,-107.320,431.990,169.895,30.888,155.860
C07832=1049.803,-107.570,431.999,169.892,30.888,155.860
C07833=1049.797,-107.820,432.009,169.890,30.887,155.860
C07834=1049.791,-108.069,432.020,169.888,30.886,155.860
C07835=1049.785,-108.319,432.029,169.886,30.886,155.860
C07836=1049.779,-108.569,432.039,169.883,30.885,155.860
C07837=1049.772,-108.818,432.049,169.881,30.885,155.860
C07838=1049.766,-109.068,432.059,169.879,30.884,155.861
C07839=1049.760,-109.317,432.068,169.877,30.884,155.861
C07840=1049.754,-109.567,432.078,169.875,30.884,155.861
C07841=1049.747,-109.817,432.088,169.872,30.883,155.861
C07842=1049.742,-110.067,432.098,169.870,30.882,155.861
C07843=1049.736,-110.317,432.107,169.869,30.882,155.861
C07844=1049.729,-110.566,432.118,169.867,30.882,155.861
C07845=1049.723,-110.816,432.127,169.864,30.881,155.861
C07846=1049.717,-111.066,432.137,169.862,30.880,155.861
C07847=1049.711,-111.316,432.146,169.860,30.880,155.861
C07848=1049.705,-111.565,432.156,169.858,30.880,155.861
C07849=1049.698,-111.815,432.165,169.855,30.879,155.861
C07850=1049.692,-112.065,432.175,169.853,30.878,155.861
C07851=1049.686,-112.314,432.185,169.851,30.878,155.861
C07852=1049.680,-112.564,432.195,169.849,30.878,155.861
C07853=1049.674,-112.814,432.205,169.846,30.877,155.861
C07854=1049.668,-113.064,432.215,169.844,30.877,155.861
C07855=1049.662,-113.314,432.224,169.842,30.877,155.861
C07856=1049.656,-113.563,432.234,169.840,30.876,155.861
C07857=1049.649,-113.813,432.243,169.838,30.875,155.861
C07858=1049.643,-114.063,432.253,169.836,30.875,155.862
C07859=1049.637,-114.313,432.262,169.834,30.875,155.862
C07860=1049.631,-114.563,432.272,169.832,30.874,155.862
C07861=1049.625,-114.812,432.282,169.829,30.874,155.862
C07862=1049.618,-115.097,432.292,169.827,30.874,155.862
C07863=1049.611,-115.383,432.303,169.824,30.873,155.862
C07864=1049.604,-115.668,432.314,169.822,30.873,155.862
C07865=1049.597,-115.953,432.325,169.819,30.872,155.862
C07866=1049.591,-116.202,432.334,169.817,30.872,155.862
C07867=1049.585,-116.452,432.344,169.815,30.871,155.862
C07868=1049.578,-116.702,432.353,169.812,30.871,155.862
C07869=1049.572,-116.952,432.363,169.810,30.870,155.862
C07870=1049.566,-117.202,432.372,169.808,30.870,155.862
C07871=1049.560,-117.451,432.382,169.806,30.870,155.862
C07872=1049.554,-117.701,432.392,169.804,30.869,155.862
C07873=1049.548,-117.951,432.401,169.802,30.869,155.863
C07874=1049.542,-118.200,432.410,169.800,30.869,155.863
C07875=1049.536,-118.450,432.419,169.798,30.868,155.863
C07876=1049.529,-118.700,432.428,169.795,30.868,155.863
C07877=1049.523,-118.950,432.438,169.793,30.868,155.863
C07878=1049.517,-119.200,432.447,169.791,30.868,155.863
C07879=1049.511,-119.449,432.457,169.789,30.868,155.863
C07880=1049.505,-119.699,432.466,169.786,30.867,155.863
C07881=1049.498,-119.949,432.476,169.784,30.867,155.863
C07882=1049.493,-120.198,432.485,169.782,30.867,155.863
C07883=1049.487,-120.448,432.494,169.780,30.866,155.863
C07884=1049.481,-120.698,432.504,169.777,30.866,155.863
C07885=1049.474,-120.948,432.513,169.775,30.866,155.864
C07886=1049.468,-121.198,432.522,169.773,30.865,155.864
C07887=1049.462,-121.447,432.531,169.771,30.865,155.864
C07888=1049.456,-121.697,432.540,169.769,30.864,155.864
C07889=1049.450,-121.947,432.550,169.767,30.865,155.864
C07890=1049.444,-122.197,432.559,169.765,30.864,155.864
C07891=1049.437,-122.446,432.568,169.763,30.864,155.864
C07892=1049.431,-122.697,432.577,169.760,30.864,155.864
C07893=1049.426,-122.946,432.586,169.758,30.863,155.864
C07894=1049.419,-123.195,432.596,169.756,30.863,155.864
C07895=1049.413,-123.445,432.606,169.754,30.863,155.864
C07896=1049.407,-123.696,432.614,169.751,30.863,155.865
C07897=1049.401,-123.944,432.623,169.749,30.863,155.865
C07898=1049.395,-124.194,432.633,169.747,30.862,155.865
C07899=1049.389,-124.444,432.642,169.744,30.862,155.865
C07900=1049.383,-124.694,432.651,169.742,30.862,155.865
C07901=1049.376,-124.944,432.660,169.740,30.862,155.865
C07902=1049.370,-125.193,432.669,169.738,30.862,155.865
C07903=1049.364,-125.443,432.678,169.735,30.861,155.865
C07904=1049.358,-125.693,432.688,169.733,30.861,155.865
C07905=1049.351,-125.943,432.697,169.732,30.861,155.865
C07906=1049.346,-126.192,432.705,169.730,30.861,155.865
C07907=1049.340,-126.442,432.715,169.727,30.860,155.866
C07908=1049.333,-126.692,432.723,169.725,30.861,155.866
C07909=1049.327,-126.942,432.732,169.723,30.860,155.866
C07910=1049.322,-127.191,432.742,169.721,30.860,155.866
C07911=1049.315,-127.441,432.750,169.718,30.860,155.866
C07912=1049.309,-127.691,432.759,169.716,30.860,155.866
C07913=1049.303,-127.940,432.769,169.714,30.860,155.866
C07914=1049.299,-128.190,432.778,169.712,30.859,155.866
C07915=1049.295,-128.440,432.789,169.710,30.858,155.866
C07916=1049.292,-128.690,432.800,169.708,30.856,155.866
C07917=1049.291,-128.940,432.811,169.706,30.853,155.866
C07918=1049.290,-129.191,432.824,169.705,30.851,155.865
C07919=1049.290,-129.441,432.837,169.703,30.847,155.865
C07920=1049.293,-129.692,432.851,169.702,30.844,155.864
C07921=1049.295,-129.942,432.865,169.700,30.840,155.864
C07922=1049.298,-130.193,432.880,169.700,30.835,155.863
C07923=1049.302,-130.443,432.896,169.699,30.830,155.862
C07924=1049.307,-130.694,432.913,169.698,30.824,155.861
C07925=1049.314,-130.944,432.929,169.698,30.819,155.860
C07926=1048.952,-130.967,432.700,169.651,30.989,155.892
C07927=1048.945,-130.717,432.684,169.652,30.995,155.893
C07928=1048.940,-130.467,432.667,169.653,31.000,155.894
C07929=1048.935,-130.216,432.652,169.654,31.006,155.895
C07930=1048.932,-129.965,432.636,169.655,31.010,155.896
C07931=1048.929,-129.715,432.623,169.656,31.015,155.896
C07932=1048.928,-129.465,432.608,169.658,31.018,155.897
C07933=1048.927,-129.215,432.595,169.659,31.022,155.897
C07934=1048.928,-128.964,432.582,169.660,31.024,155.898
C07935=1048.930,-128.714,432.571,169.662,31.027,155.898
C07936=1048.932,-128.464,432.560,169.664,31.028,155.898
C07937=1048.935,-128.214,432.550,169.666,31.030,155.898
C07938=1048.940,-127.964,432.540,169.668,31.031,155.898
C07939=1048.946,-127.715,432.530,169.670,31.031,155.898
C07940=1048.952,-127.465,432.521,169.673,31.031,155.898
C07941=1048.958,-127.215,432.512,169.675,31.031,155.898
C07942=1048.964,-126.966,432.503,169.677,31.031,155.898
C07943=1048.970,-126.715,432.494,169.679,31.031,155.898
C07944=1048.976,-126.466,432.485,169.681,31.031,155.898
C07945=1048.983,-126.217,432.476,169.683,31.032,155.898
C07946=1048.989,-125.966,432.467,169.685,31.031,155.897
C07947=1048.995,-125.716,432.458,169.688,31.032,155.897
C07948=1049.001,-125.468,432.449,169.690,31.032,155.897
C07949=1049.007,-125.217,432.440,169.692,31.032,155.897
C07950=1049.013,-124.967,432.431,169.695,31.032,155.897
C07951=1049.019,-124.718,432.421,169.697,31.033,155.897
C07952=1049.026,-124.467,432.413,169.699,31.033,155.897
C07953=1049.032,-124.218,432.404,169.701,31.032,155.897
C07954=1049.038,-123.969,432.394,169.704,31.033,155.897
C07955=1049.044,-123.718,432.385,169.706,31.033,155.897
C07956=1049.050,-123.469,432.376,169.708,31.034,155.897
C07957=1049.056,-123.220,432.367,169.710,31.034,155.896
C07958=1049.062,-122.970,432.358,169.713,31.034,155.896
C07959=1049.068,-122.719,432.349,169.715,31.034,155.896
C07960=1049.074,-122.470,432.339,169.717,31.034,155.896
C07961=1049.080,-122.220,432.330,169.719,31.035,155.896
C07962=1049.087,-121.971,432.321,169.721,31.035,155.896
C07963=1049.093,-121.721,432.312,169.723,31.035,155.896
C07964=1049.099,-121.471,432.303,169.725,31.036,155.896
C07965=1049.105,-121.221,432.293,169.728,31.035,155.896
C07966=1049.111,-120.971,432.284,169.730,31.036,155.896
C07967=1049.117,-120.722,432.274,169.732,31.036,155.896
C07968=1049.123,-120.472,432.265,169.734,31.036,155.895
C07969=1049.129,-120.222,432.256,169.737,31.037,155.895
C07970=1049.136,-119.972,432.247,169.739,31.037,155.895
C07971=1049.142,-119.723,432.237,169.741,31.037,155.895
C07972=1049.148,-119.473,432.228,169.743,31.038,155.895
C07973=1049.154,-119.223,432.218,169.746,31.038,155.895
C07974=1049.160,-118.974,432.209,169.748,31.038,155.895
C07975=1049.166,-118.723,432.200,169.750,31.039,155.895
C07976=1049.172,-118.474,432.191,169.752,31.038,155.895
C07977=1049.178,-118.224,432.181,169.755,31.039,155.895
C07978=1049.185,-117.974,432.172,169.756,31.039,155.895
C07979=1049.191,-117.725,432.162,169.758,31.039,155.895
C07980=1049.197,-117.475,432.153,169.761,31.040,155.894
C07981=1049.203,-117.225,432.143,169.763,31.040,155.894
C07982=1049.209,-116.976,432.134,169.765,31.040,155.894
C07983=1049.215,-116.726,432.125,169.767,31.041,155.894
C07984=1049.221,-116.476,432.115,169.770,31.041,155.894
C07985=1049.227,-116.227,432.105,169.772,31.041,155.894
C07986=1049.234,-115.977,432.096,169.774,31.042,155.894
C07987=1049.241,-115.692,432.085,169.777,31.042,155.894
C07988=1049.247,-115.406,432.075,169.779,31.043,155.894
C07989=1049.255,-115.120,432.064,169.782,31.043,155.894
C07990=1049.262,-114.835,432.053,169.784,31.044,155.894
C07991=1049.268,-114.585,432.044,169.787,31.044,155.894
C07992=1049.274,-114.336,432.034,169.789,31.045,155.894
C07993=1049.280,-114.086,432.024,169.790,31.045,155.894
C07994=1049.286,-113.836,432.015,169.792,31.045,155.894
C07995=1049.292,-113.587,432.004,169.795,31.046,155.893
C07996=1049.298,-113.337,431.994,169.797,31.046,155.893
C07997=1049.304,-113.088,431.985,169.799,31.046,155.893
C07998=1049.310,-112.838,431.976,169.801,31.047,155.893
C07999=1049.316,-112.588,431.966,169.804,31.048,155.893
C08000=1049.322,-112.338,431.957,169.806,31.048,155.893
C08001=1049.329,-112.088,431.947,169.808,31.048,155.893
C08002=1049.335,-111.839,431.937,169.810,31.049,155.893
C08003=1049.341,-111.589,431.928,169.813,31.049,155.893
C08004=1049.347,-111.339,431.918,169.815,31.049,155.893
C08005=1049.354,-111.090,431.908,169.817,31.050,155.893
C08006=1049.360,-110.840,431.898,169.819,31.050,155.893
C08007=1049.365,-110.590,431.888,169.822,31.051,155.893
C08008=1049.371,-110.340,431.879,169.823,31.051,155.893
C08009=1049.378,-110.090,431.869,169.825,31.052,155.893
C08010=1049.384,-109.841,431.860,169.827,31.052,155.893
C08011=1049.390,-109.591,431.849,169.830,31.053,155.893
C08012=1049.396,-109.342,431.840,169.832,31.053,155.893
C08013=1049.403,-109.092,431.830,169.834,31.053,155.893
C08014=1049.409,-108.842,431.821,169.836,31.054,155.893
C08015=1049.415,-108.592,431.811,169.839,31.055,155.893
C08016=1049.421,-108.343,431.800,169.841,31.055,155.892
C08017=1049.427,-108.093,431.791,169.843,31.055,155.892
C08018=1049.433,-107.843,431.781,169.845,31.056,155.892
C08019=1049.440,-107.593,431.771,169.848,31.057,155.892
C08020=1049.446,-107.343,431.761,169.850,31.057,155.892
C08021=1049.452,-107.094,431.751,169.852,31.057,155.892
C08022=1049.458,-106.844,431.741,169.853,31.058,155.892
C08023=1049.464,-106.594,431.731,169.855,31.059,155.892
C08024=1049.470,-106.345,431.721,169.858,31.059,155.892
C08025=1049.477,-106.095,431.712,169.860,31.060,155.892
C08026=1049.482,-105.845,431.701,169.862,31.060,155.892
C08027=1049.489,-105.595,431.691,169.864,31.061,155.892
C08028=1049.495,-105.346,431.682,169.867,31.062,155.892
C08029=1049.501,-105.096,431.672,169.869,31.062,155.892
C08030=1049.507,-104.846,431.661,169.871,31.063,155.892
C08031=1049.513,-104.597,431.652,169.873,31.063,155.892
C08032=1049.519,-104.347,431.642,169.876,31.064,155.892
C08033=1049.525,-104.098,431.632,169.878,31.065,155.892
C08034=1049.532,-103.847,431.621,169.880,31.065,155.892
C08035=1049.538,-103.597,431.612,169.882,31.066,155.892
C08036=1049.544,-103.348,431.601,169.883,31.066,155.892
C08037=1049.550,-103.098,431.591,169.886,31.066,155.892
C08038=1049.556,-102.849,431.581,169.888,31.067,155.892
C08039=1049.562,-102.599,431.571,169.890,31.068,155.892
C08040=1049.568,-102.349,431.560,169.892,31.069,155.892
C08041=1049.574,-102.099,431.551,169.895,31.069,155.892
C08042=1049.580,-101.850,431.541,169.897,31.070,155.892
C08043=1049.587,-101.599,431.530,169.899,31.070,155.892
C08044=1049.593,-101.350,431.521,169.901,31.071,155.892
C08045=1049.599,-101.101,431.510,169.903,31.071,155.892
C08046=1049.605,-100.850,431.500,169.906,31.073,155.892
C08047=1049.611,-100.601,431.490,169.908,31.073,155.892
C08048=1049.617,-100.351,431.480,169.910,31.074,155.892
C08049=1049.624,-100.101,431.469,169.911,31.074,155.892
C08050=1049.630,-99.851,431.459,169.914,31.075,155.892
C08051=1049.637,-99.565,431.448,169.916,31.075,155.892
C08052=1049.644,-99.279,431.436,169.919,31.076,155.892
C08053=1049.652,-98.993,431.424,169.921,31.077,155.892
C08054=1049.658,-98.706,431.412,169.924,31.078,155.892
C08055=1049.665,-98.456,431.402,169.926,31.079,155.892
C08056=1049.671,-98.207,431.392,169.928,31.079,155.892
C08057=1049.677,-97.957,431.382,169.930,31.080,155.892
C08058=1049.683,-97.708,431.371,169.933,31.080,155.892
C08059=1049.689,-97.458,431.361,169.935,31.081,155.892
C08060=1049.696,-97.208,431.351,169.937,31.082,155.892
C08061=1049.701,-96.958,431.340,169.938,31.083,155.892
C08062=1049.707,-96.708,431.330,169.940,31.083,155.892
C08063=1049.713,-96.459,431.319,169.943,31.085,155.892
C08064=1049.720,-96.210,431.309,169.945,31.085,155.892
C08065=1049.726,-95.959,431.299,169.947,31.086,155.892
C08066=1049.732,-95.710,431.288,169.949,31.087,155.892
C08067=1049.738,-95.460,431.277,169.951,31.087,155.892
C08068=1049.743,-95.210,431.267,169.954,31.088,155.892
C08069=1049.750,-94.961,431.257,169.956,31.089,155.892
C08070=1049.756,-94.711,431.246,169.958,31.090,155.892
C08071=1049.763,-94.461,431.235,169.960,31.090,155.892
C08072=1049.768,-94.211,431.225,169.962,31.091,155.892
C08073=1049.774,-93.962,431.214,169.964,31.092,155.892
C08074=1049.780,-93.713,431.204,169.966,31.093,155.892
C08075=1049.787,-93.462,431.193,169.968,31.093,155.892
C08076=1049.792,-93.212,431.183,169.970,31.094,155.892
C08077=1049.799,-92.963,431.172,169.972,31.095,155.892
C08078=1049.804,-92.714,431.162,169.974,31.096,155.892
C08079=1049.811,-92.464,431.151,169.977,31.097,155.892
C08080=1049.817,-92.214,431.141,169.979,31.097,155.892
C08081=1049.823,-91.964,431.130,169.981,31.098,155.892
C08082=1049.830,-91.714,431.119,169.983,31.099,155.892
C08083=1049.835,-91.465,431.108,169.985,31.100,155.892
C08084=1049.842,-91.216,431.098,169.987,31.101,155.892
C08085=1049.847,-90.966,431.088,169.989,31.102,155.892
C08086=1049.854,-90.715,431.077,169.991,31.103,155.892
C08087=1049.860,-90.466,431.066,169.993,31.103,155.892
C08088=1049.866,-90.217,431.055,169.995,31.104,155.892
C08089=1049.872,-89.966,431.044,169.998,31.105,155.892
C08090=1049.879,-89.717,431.034,170.000,31.106,155.892
C08091=1049.884,-89.468,431.023,170.002,31.107,155.892
C08092=1049.890,-89.217,431.013,170.004,31.108,155.892
C08093=1049.897,-88.968,431.002,170.006,31.108,155.892
C08094=1049.903,-88.718,430.991,170.008,31.109,155.892
C08095=1049.909,-88.468,430.980,170.011,31.110,155.892
C08096=1049.915,-88.219,430.970,170.012,31.111,155.892
C08097=1049.921,-87.969,430.959,170.014,31.112,155.892
C08098=1049.928,-87.719,430.948,170.016,31.113,155.892
C08099=1049.934,-87.470,430.937,170.018,31.113,155.892
C08100=1049.940,-87.220,430.926,170.021,31.115,155.892
C08101=1049.946,-86.970,430.915,170.023,31.115,155.892
C08102=1049.953,-86.721,430.905,170.025,31.116,155.892
C08103=1049.959,-86.471,430.894,170.027,31.117,155.893
C08104=1049.965,-86.222,430.883,170.029,31.118,155.893
C08105=1049.971,-85.972,430.873,170.031,31.119,155.893
C08106=1049.977,-85.722,430.861,170.034,31.120,155.893
C08107=1049.983,-85.473,430.851,170.036,31.120,155.893
C08108=1049.990,-85.223,430.840,170.037,31.121,155.893
C08109=1049.996,-84.973,430.829,170.039,31.122,155.893
C08110=1050.002,-84.723,430.818,170.041,31.123,155.893
C08111=1050.009,-84.474,430.807,170.043,31.124,155.893
C08112=1050.015,-84.224,430.797,170.046,31.125,155.893
C08113=1050.021,-83.974,430.785,170.048,31.126,155.893
C08114=1050.027,-83.725,430.774,170.050,31.127,155.893
C08115=1050.034,-83.441,430.762,170.052,31.128,155.893
C08116=1050.041,-83.156,430.750,170.055,31.129,155.893
C08117=1050.049,-82.872,430.737,170.057,31.130,155.893
C08118=1050.056,-82.588,430.725,170.059,31.131,155.893
C08119=1050.062,-82.338,430.714,170.061,31.132,155.893
C08120=1050.069,-82.088,430.703,170.063,31.133,155.893
C08121=1050.074,-81.839,430.692,170.065,31.134,155.893
C08122=1050.081,-81.589,430.681,170.068,31.135,155.893
C08123=1050.087,-81.340,430.670,170.070,31.136,155.893
C08124=1050.094,-81.090,430.659,170.072,31.137,155.893
C08125=1050.100,-80.840,430.648,170.074,31.138,155.893
C08126=1050.106,-80.590,430.637,170.076,31.138,155.893
C08127=1050.112,-80.341,430.626,170.078,31.139,155.893
C08128=1050.119,-80.091,430.615,170.080,31.140,155.894
C08129=1050.125,-79.842,430.604,170.082,31.141,155.894
C08130=1050.131,-79.592,430.592,170.084,31.142,155.894
C08131=1050.137,-79.342,430.582,170.086,31.144,155.894
C08132=1050.143,-79.092,430.570,170.088,31.145,155.894
C08133=1050.149,-78.843,430.559,170.090,31.146,155.894
C08134=1050.156,-78.593,430.547,170.092,31.147,155.894
C08135=1050.161,-78.344,430.537,170.095,31.148,155.894
C08136=1050.168,-78.093,430.525,170.097,31.149,155.894
C08137=1050.173,-77.844,430.514,170.099,31.150,155.894
C08138=1050.180,-77.594,430.503,170.101,31.151,155.894
C08139=1050.187,-77.345,430.492,170.103,31.152,155.894
C08140=1050.193,-77.095,430.481,170.104,31.153,155.894
C08141=1050.199,-76.846,430.469,170.106,31.154,155.894
C08142=1050.205,-76.596,430.458,170.108,31.155,155.895
C08143=1050.211,-76.346,430.447,170.111,31.156,155.895
C08144=1050.218,-76.097,430.435,170.113,31.157,155.895
C08145=1050.223,-75.847,430.424,170.115,31.158,155.895
C08146=1050.230,-75.597,430.413,170.117,31.159,155.895
C08147=1050.236,-75.348,430.401,170.119,31.161,155.895
C08148=1050.242,-75.098,430.390,170.121,31.161,155.895
C08149=1050.248,-74.848,430.379,170.123,31.162,155.895
C08150=1050.254,-74.599,430.368,170.125,31.163,155.895
C08151=1050.261,-74.349,430.356,170.127,31.165,155.895
C08152=1050.267,-74.100,430.345,170.129,31.166,155.895
C08153=1050.273,-73.850,430.333,170.131,31.167,155.895
C08154=1050.279,-73.599,430.322,170.133,31.168,155.895
C08155=1050.285,-73.350,430.310,170.135,31.169,155.895
C08156=1050.291,-73.100,430.299,170.137,31.170,155.896
C08157=1050.297,-72.851,430.287,170.139,31.172,155.896
C08158=1050.304,-72.601,430.276,170.142,31.173,155.896
C08159=1050.309,-72.352,430.264,170.144,31.174,155.896
C08160=1050.315,-72.102,430.252,170.145,31.175,155.896
C08161=1050.321,-71.853,430.241,170.147,31.176,155.896
C08162=1050.328,-71.603,430.230,170.149,31.178,155.896
C08163=1050.334,-71.353,430.217,170.151,31.179,155.896
C08164=1050.339,-71.103,430.206,170.153,31.180,155.896
C08165=1050.346,-70.854,430.194,170.155,31.181,155.896
C08166=1050.352,-70.604,430.183,170.157,31.183,155.897
C08167=1050.358,-70.354,430.171,170.159,31.183,155.897
C08168=1050.363,-70.105,430.160,170.162,31.184,155.897
C08169=1050.370,-69.855,430.148,170.164,31.186,155.897
C08170=1050.376,-69.605,430.137,170.165,31.187,155.897
C08171=1050.382,-69.356,430.125,170.167,31.188,155.897
C08172=1050.388,-69.106,430.113,170.169,31.189,155.897
C08173=1050.395,-68.856,430.101,170.171,31.191,155.897
C08174=1050.401,-68.607,430.090,170.173,31.192,155.897
C08175=1050.406,-68.357,430.078,170.175,31.193,155.897
C08176=1050.413,-68.107,430.066,170.177,31.194,155.897
C08177=1050.419,-67.858,430.054,170.179,31.196,155.898
C08178=1050.425,-67.608,430.043,170.182,31.197,155.898
C08179=1050.432,-67.326,430.029,170.184,31.198,155.898
C08180=1050.439,-67.045,430.016,170.185,31.200,155.898
C08181=1050.445,-66.762,430.003,170.188,31.201,155.898
C08182=1050.453,-66.480,429.989,170.190,31.202,155.898
C08183=1050.459,-66.231,429.978,170.192,31.203,155.898
C08184=1050.465,-65.981,429.967,170.194,31.205,155.898
C08185=1050.471,-65.731,429.954,170.196,31.206,155.899
C08186=1050.477,-65.482,429.942,170.198,31.207,155.899
C08187=1050.483,-65.232,429.931,170.200,31.209,155.899
C08188=1050.490,-64.983,429.919,170.203,31.210,155.899
C08189=1050.496,-64.733,429.907,170.204,31.211,155.899
C08190=1050.502,-64.484,429.895,170.206,31.212,155.899
C08191=1050.508,-64.234,429.884,170.208,31.214,155.899
C08192=1050.514,-63.984,429.871,170.210,31.215,155.899
C08193=1050.520,-63.735,429.860,170.212,31.216,155.899
C08194=1050.527,-63.485,429.848,170.214,31.217,155.899
C08195=1050.532,-63.235,429.836,170.216,31.219,155.900
C08196=1050.539,-62.985,429.824,170.218,31.220,155.900
C08197=1050.545,-62.736,429.812,170.220,31.221,155.900
C08198=1050.551,-62.486,429.800,170.222,31.223,155.900
C08199=1050.558,-62.237,429.788,170.224,31.224,155.900
C08200=1050.564,-61.987,429.777,170.226,31.225,155.900
C08201=1050.570,-61.737,429.764,170.228,31.226,155.900
C08202=1050.576,-61.488,429.752,170.230,31.228,155.900
C08203=1050.583,-61.238,429.740,170.232,31.229,155.900
C08204=1050.588,-60.988,429.728,170.234,31.230,155.901
C08205=1050.595,-60.739,429.716,170.236,31.232,155.901
C08206=1050.601,-60.489,429.705,170.238,31.233,155.901
C08207=1050.607,-60.239,429.692,170.240,31.234,155.901
C08208=1050.613,-59.990,429.681,170.242,31.235,155.901
C08209=1050.620,-59.740,429.669,170.243,31.237,155.901
C08210=1050.626,-59.490,429.656,170.245,31.238,155.901
C08211=1050.633,-59.241,429.644,170.247,31.239,155.901
C08212=1050.639,-58.992,429.632,170.249,31.240,155.902
C08213=1050.645,-58.742,429.620,170.252,31.242,155.902
C08214=1050.651,-58.493,429.608,170.254,31.243,155.902
C08215=1050.657,-58.242,429.596,170.256,31.245,155.902
C08216=1050.663,-57.992,429.584,170.258,31.245,155.902
C08217=1050.670,-57.743,429.572,170.260,31.247,155.902
C08218=1050.676,-57.493,429.560,170.261,31.249,155.902
C08219=1050.683,-57.243,429.548,170.263,31.249,155.902
C08220=1050.689,-56.995,429.536,170.265,31.251,155.903
C08221=1050.695,-56.745,429.524,170.267,31.252,155.903
C08222=1050.701,-56.495,429.512,170.269,31.253,155.903
C08223=1050.707,-56.245,429.499,170.271,31.255,155.903
C08224=1050.714,-55.996,429.487,170.273,31.256,155.903
C08225=1050.720,-55.746,429.475,170.275,31.257,155.903
C08226=1050.726,-55.496,429.463,170.277,31.259,155.903
C08227=1050.733,-55.247,429.451,170.279,31.260,155.903
C08228=1050.740,-54.997,429.439,170.281,31.261,155.904
C08229=1050.746,-54.747,429.426,170.283,31.263,155.904
C08230=1050.752,-54.498,429.414,170.285,31.264,155.904
C08231=1050.758,-54.248,429.402,170.287,31.265,155.904
C08232=1050.764,-54.000,429.389,170.289,31.267,155.904
C08233=1050.770,-53.750,429.377,170.291,31.268,155.904
C08234=1050.777,-53.500,429.365,170.293,31.269,155.904
C08235=1050.784,-53.250,429.353,170.295,31.271,155.904
C08236=1050.790,-53.001,429.340,170.297,31.272,155.905
C08237=1050.796,-52.751,429.328,170.299,31.273,155.905
C08238=1050.802,-52.501,429.316,170.300,31.275,155.905
C08239=1050.809,-52.252,429.304,170.302,31.276,155.905
C08240=1050.815,-52.002,429.292,170.304,31.277,155.905
C08241=1050.821,-51.752,429.279,170.306,31.279,155.905
C08242=1050.828,-51.503,429.267,170.308,31.280,155.905
C08243=1050.835,-51.222,429.253,170.311,31.282,155.906
C08244=1050.843,-50.942,429.239,170.313,31.283,155.906
C08245=1050.849,-50.661,429.225,170.315,31.285,155.906
C08246=1050.857,-50.380,429.211,170.318,31.287,155.906
C08247=1050.863,-50.130,429.199,170.319,31.288,155.906
C08248=1050.869,-49.880,429.186,170.321,31.289,155.906
C08249=1050.875,-49.631,429.174,170.323,31.291,155.906
C08250=1050.881,-49.382,429.161,170.325,31.292,155.907
C08251=1050.887,-49.132,429.149,170.327,31.294,155.907
C08252=1050.893,-48.883,429.136,170.329,31.295,155.907
C08253=1050.899,-48.633,429.124,170.331,31.297,155.907
C08254=1050.905,-48.383,429.110,170.333,31.298,155.907
C08255=1050.912,-48.134,429.098,170.335,31.300,155.907
C08256=1050.918,-47.884,429.086,170.336,31.301,155.908
C08257=1050.924,-47.635,429.072,170.338,31.303,155.908
C08258=1050.930,-47.385,429.060,170.340,31.304,155.908
C08259=1050.937,-47.135,429.048,170.342,31.306,155.908
C08260=1050.943,-46.886,429.035,170.344,31.307,155.908
C08261=1050.949,-46.636,429.022,170.346,31.309,155.908
C08262=1050.955,-46.386,429.010,170.348,31.310,155.909
C08263=1050.962,-46.137,428.997,170.350,31.312,155.909
C08264=1050.968,-45.887,428.984,170.352,31.313,155.909
C08265=1050.974,-45.638,428.972,170.353,31.315,155.909
C08266=1050.980,-45.388,428.959,170.355,31.316,155.909
C08267=1050.986,-45.139,428.947,170.357,31.318,155.909
C08268=1050.993,-44.889,428.933,170.359,31.319,155.910
C08269=1050.999,-44.640,428.921,170.361,31.321,155.910
C08270=1051.004,-44.390,428.908,170.363,31.322,155.910
C08271=1051.011,-44.140,428.895,170.365,31.324,155.910
C08272=1051.017,-43.891,428.883,170.367,31.325,155.910
C08273=1051.024,-43.641,428.869,170.369,31.327,155.910
C08274=1051.030,-43.391,428.857,170.371,31.329,155.911
C08275=1051.036,-43.142,428.843,170.372,31.330,155.911
C08276=1051.042,-42.892,428.831,170.374,31.332,155.911
C08277=1051.049,-42.642,428.819,170.376,31.333,155.911
C08278=1051.055,-42.393,428.806,170.378,31.335,155.911
C08279=1051.061,-42.143,428.793,170.380,31.336,155.911
C08280=1051.067,-41.894,428.780,170.382,31.338,155.912
C08281=1051.073,-41.644,428.767,170.384,31.339,155.912
C08282=1051.079,-41.395,428.754,170.386,31.341,155.912
C08283=1051.086,-41.145,428.742,170.388,31.342,155.912
C08284=1051.093,-40.895,428.728,170.389,31.344,155.912
C08285=1051.099,-40.645,428.716,170.391,31.345,155.912
C08286=1051.105,-40.396,428.703,170.393,31.347,155.913
C08287=1051.111,-40.147,428.689,170.395,31.348,155.913
C08288=1051.118,-39.897,428.677,170.397,31.350,155.913
C08289=1051.124,-39.648,428.664,170.399,31.351,155.913
C08290=1051.130,-39.398,428.652,170.401,31.353,155.913
C08291=1051.137,-39.148,428.638,170.403,31.354,155.913
C08292=1051.143,-38.898,428.625,170.405,31.356,155.914
C08293=1051.149,-38.649,428.612,170.406,31.357,155.914
C08294=1051.155,-38.400,428.599,170.408,31.359,155.914
C08295=1051.161,-38.150,428.586,170.410,31.361,155.914
C08296=1051.167,-37.900,428.573,170.412,31.362,155.914
C08297=1051.173,-37.651,428.560,170.414,31.364,155.915
C08298=1051.180,-37.401,428.547,170.415,31.365,155.915
C08299=1051.186,-37.151,428.534,170.417,31.367,155.915
C08300=1051.192,-36.902,428.520,170.419,31.369,155.915
C08301=1051.198,-36.652,428.508,170.421,31.370,155.915
C08302=1051.204,-36.403,428.494,170.422,31.372,155.916
C08303=1051.211,-36.154,428.481,170.424,31.374,155.916
C08304=1051.216,-35.904,428.469,170.426,31.375,155.916
C08305=1051.223,-35.654,428.455,170.428,31.377,155.916
C08306=1051.230,-35.405,428.442,170.430,31.379,155.916
C08307=1051.237,-35.125,428.427,170.432,31.380,155.916
C08308=1051.243,-34.844,428.412,170.435,31.382,155.917
C08309=1051.250,-34.563,428.398,170.437,31.384,155.917
C08310=1051.257,-34.283,428.383,170.439,31.386,155.917
C08311=1051.263,-34.034,428.370,170.440,31.388,155.917
C08312=1051.269,-33.785,428.356,170.442,31.389,155.917
C08313=1051.276,-33.535,428.343,170.444,31.391,155.918
C08314=1051.282,-33.285,428.330,170.446,31.393,155.918
C08315=1051.288,-33.036,428.317,170.448,31.394,155.918
C08316=1051.294,-32.786,428.304,170.450,31.396,155.918
C08317=1051.300,-32.537,428.290,170.452,31.397,155.918
C08318=1051.307,-32.287,428.276,170.454,31.399,155.919
C08319=1051.313,-32.038,428.263,170.455,31.401,155.919
C08320=1051.319,-31.788,428.250,170.456,31.402,155.919
C08321=1051.325,-31.538,428.237,170.458,31.404,155.919
C08322=1051.332,-31.288,428.223,170.460,31.406,155.920
C08323=1051.338,-31.039,428.210,170.462,31.407,155.920
C08324=1051.344,-30.790,428.197,170.464,31.409,155.920
C08325=1051.350,-30.541,428.183,170.466,31.410,155.920
C08326=1051.357,-30.291,428.170,170.468,31.413,155.920
C08327=1051.362,-30.041,428.157,170.470,31.414,155.921
C08328=1051.369,-29.791,428.143,170.472,31.416,155.921
C08329=1051.375,-29.541,428.130,170.473,31.417,155.921
C08330=1051.382,-29.292,428.117,170.475,31.419,155.921
C08331=1051.388,-29.043,428.103,170.477,31.421,155.921
C08332=1051.395,-28.793,428.090,170.479,31.422,155.921
C08333=1051.401,-28.544,428.076,170.481,31.424,155.922
C08334=1051.407,-28.294,428.063,170.483,31.426,155.922
C08335=1051.413,-28.045,428.049,170.485,31.427,155.922
C08336=1051.419,-27.795,428.036,170.486,31.429,155.922
C08337=1051.426,-27.546,428.022,170.488,31.431,155.923
C08338=1051.432,-27.296,428.009,170.489,31.432,155.923
C08339=1051.439,-27.046,427.995,170.491,31.434,155.923
C08340=1051.445,-26.797,427.982,170.493,31.435,155.923
C08341=1051.450,-26.547,427.968,170.495,31.437,155.923
C08342=1051.457,-26.297,427.955,170.497,31.439,155.924
C08343=1051.463,-26.048,427.941,170.499,31.441,155.924
C08344=1051.469,-25.799,427.927,170.501,31.443,155.924
C08345=1051.476,-25.549,427.914,170.503,31.445,155.924
C08346=1051.481,-25.299,427.900,170.505,31.446,155.924
C08347=1051.487,-25.050,427.887,170.506,31.448,155.925
C08348=1051.494,-24.800,427.873,170.507,31.450,155.925
C08349=1051.500,-24.550,427.859,170.509,31.451,155.925
C08350=1051.506,-24.301,427.846,170.511,31.453,155.925
C08351=1051.513,-24.051,427.832,170.513,31.455,155.926
C08352=1051.518,-23.802,427.818,170.515,31.457,155.926
C08353=1051.525,-23.553,427.804,170.517,31.458,155.926
C08354=1051.531,-23.303,427.791,170.519,31.460,155.926
C08355=1051.537,-23.053,427.777,170.521,31.462,155.926
C08356=1051.543,-22.804,427.764,170.523,31.464,155.927
C08357=1051.549,-22.554,427.749,170.524,31.466,155.927
C08358=1051.555,-22.304,427.736,170.525,31.467,155.927
C08359=1051.563,-22.055,427.722,170.527,31.469,155.927
C08360=1051.568,-21.806,427.708,170.529,31.471,155.928
C08361=1051.574,-21.556,427.695,170.531,31.473,155.928
C08362=1051.580,-21.306,427.680,170.533,31.474,155.928
C08363=1051.587,-21.057,427.667,170.535,31.476,155.928
C08364=1051.594,-20.807,427.653,170.537,31.478,155.928
C08365=1051.599,-20.558,427.639,170.539,31.479,155.929
C08366=1051.605,-20.309,427.626,170.540,31.482,155.929
C08367=1051.611,-20.058,427.611,170.542,31.483,155.929
C08368=1051.618,-19.809,427.598,170.543,31.485,155.929
C08369=1051.625,-19.560,427.584,170.545,31.487,155.930
C08370=1051.630,-19.310,427.570,170.547,31.489,155.930
C08371=1051.637,-19.029,427.554,170.549,31.490,155.930
C08372=1051.645,-18.748,427.539,170.551,31.492,155.930
C08373=1051.652,-18.467,427.523,170.554,31.495,155.931
C08374=1051.659,-18.186,427.508,170.555,31.497,155.931
C08375=1051.665,-17.937,427.494,170.557,31.498,155.931
C08376=1051.671,-17.687,427.479,170.558,31.500,155.931
C08377=1051.678,-17.438,427.466,170.560,31.502,155.931
C08378=1051.684,-17.188,427.452,170.562,31.504,155.932
C08379=1051.690,-16.939,427.438,170.564,31.505,155.932
C08380=1051.696,-16.689,427.424,170.566,31.507,155.932
C08381=1051.702,-16.439,427.410,170.568,31.509,155.932
C08382=1051.709,-16.190,427.395,170.570,31.511,155.933
C08383=1051.715,-15.940,427.382,170.572,31.512,155.933
C08384=1051.722,-15.690,427.369,170.573,31.515,155.933
C08385=1051.728,-15.442,427.354,170.574,31.516,155.933
C08386=1051.734,-15.192,427.340,170.576,31.518,155.934
C08387=1051.740,-14.943,427.326,170.578,31.520,155.934
C08388=1051.746,-14.692,427.312,170.580,31.522,155.934
C08389=1051.752,-14.443,427.298,170.582,31.523,155.934
C08390=1051.759,-14.193,427.283,170.584,31.525,155.935
C08391=1051.764,-13.944,427.269,170.586,31.527,155.935
C08392=1051.771,-13.694,427.255,170.587,31.529,155.935
C08393=1051.777,-13.445,427.241,170.588,31.531,155.935
C08394=1051.783,-13.195,427.226,170.590,31.533,155.936
C08395=1051.790,-12.946,427.213,170.592,31.534,155.936
C08396=1051.796,-12.696,427.198,170.594,31.537,155.936
C08397=1051.801,-12.447,427.184,170.596,31.538,155.936
C08398=1051.809,-12.197,427.170,170.598,31.540,155.936
C08399=1051.814,-11.948,427.156,170.599,31.542,155.937
C08400=1051.820,-11.698,427.141,170.601,31.544,155.937
C08401=1051.827,-11.449,427.128,170.603,31.546,155.937
C08402=1051.833,-11.199,427.113,170.604,31.548,155.938
C08403=1051.838,-10.950,427.099,170.606,31.549,155.938
C08404=1051.846,-10.700,427.085,170.608,31.551,155.938
C08405=1051.851,-10.451,427.071,170.610,31.553,155.938
C08406=1051.857,-10.201,427.056,170.611,31.555,155.938
C08407=1051.865,-9.952,427.041,170.613,31.557,155.939
C08408=1051.870,-9.702,427.028,170.615,31.559,155.939
C08409=1051.876,-9.453,427.013,170.617,31.561,155.939
C08410=1051.882,-9.203,426.999,170.619,31.563,155.940
C08411=1051.889,-8.954,426.984,170.620,31.564,155.940
C08412=1051.895,-8.705,426.970,170.621,31.566,155.940
C08413=1051.901,-8.454,426.956,170.623,31.568,155.940
C08414=1051.908,-8.205,426.941,170.625,31.570,155.940
C08415=1051.913,-7.955,426.927,170.627,31.572,155.941
C08416=1051.920,-7.706,426.912,170.629,31.574,155.941
C08417=1051.926,-7.457,426.899,170.631,31.576,155.941
C08418=1051.932,-7.207,426.884,170.632,31.578,155.942
C08419=1051.939,-6.957,426.869,170.634,31.579,155.942
C08420=1051.945,-6.708,426.855,170.636,31.581,155.942
C08421=1051.951,-6.458,426.841,170.637,31.583,155.942
C08422=1051.957,-6.209,426.827,170.639,31.585,155.942
C08423=1051.964,-5.960,426.812,170.641,31.587,155.943
C08424=1051.970,-5.709,426.797,170.642,31.589,155.943
C08425=1051.976,-5.461,426.783,170.644,31.590,155.943
C08426=1051.983,-5.211,426.768,170.646,31.592,155.943
C08427=1051.989,-4.961,426.753,170.648,31.595,155.944
C08428=1051.995,-4.712,426.740,170.650,31.596,155.944
C08429=1052.002,-4.463,426.725,170.652,31.598,155.944
C08430=1052.008,-4.213,426.710,170.652,31.600,155.945
C08431=1052.014,-3.964,426.696,170.654,31.602,155.945
C08432=1052.021,-3.714,426.682,170.656,31.604,155.945
C08433=1052.027,-3.464,426.667,170.658,31.606,155.945
C08434=1052.033,-3.215,426.653,170.660,31.607,155.945
C08435=1052.040,-2.932,426.636,170.662,31.610,155.946
C08436=1052.047,-2.650,426.620,170.664,31.612,155.946
C08437=1052.054,-2.367,426.602,170.666,31.614,155.946
C08438=1052.061,-2.085,426.586,170.668,31.616,155.947
C08439=1052.067,-1.835,426.571,170.669,31.618,155.947
C08440=1052.073,-1.586,426.556,170.671,31.621,155.947
C08441=1052.079,-1.336,426.542,170.672,31.622,155.948
C08442=1052.085,-1.087,426.527,170.674,31.625,155.948
C08443=1052.091,-0.837,426.512,170.676,31.626,155.948
C08444=1052.098,-0.588,426.498,170.678,31.628,155.948
C08445=1052.103,-0.338,426.482,170.680,31.630,155.949
C08446=1052.109,-0.089,426.467,170.681,31.632,155.949
C08447=1052.115,0.161,426.452,170.683,31.634,155.949
C08448=1052.121,0.410,426.438,170.685,31.636,155.950
C08449=1052.127,0.660,426.423,170.686,31.639,155.950
C08450=1052.134,0.909,426.408,170.687,31.640,155.950
C08451=1052.140,1.159,426.393,170.689,31.642,155.950
C08452=1052.146,1.408,426.378,170.691,31.644,155.951
C08453=1052.152,1.658,426.364,170.693,31.646,155.951
C08454=1052.159,1.907,426.349,170.695,31.648,155.951
C08455=1052.165,2.156,426.334,170.696,31.650,155.951
C08456=1052.171,2.406,426.319,170.698,31.652,155.952
C08457=1052.177,2.655,426.304,170.700,31.654,155.952
C08458=1052.184,2.905,426.289,170.701,31.656,155.952
C08459=1052.190,3.154,426.275,170.703,31.658,155.953
C08460=1052.196,3.404,426.260,170.704,31.660,155.953
C08461=1052.202,3.653,426.245,170.706,31.662,155.953
C08462=1052.207,3.903,426.230,170.708,31.664,155.953
C08463=1052.214,4.152,426.215,170.710,31.666,155.954
C08464=1052.220,4.402,426.200,170.712,31.668,155.954
C08465=1052.226,4.652,426.185,170.713,31.670,155.954
C08466=1052.233,4.901,426.170,170.715,31.672,155.954
C08467=1052.239,5.150,426.155,170.717,31.674,155.955
C08468=1052.245,5.400,426.140,170.718,31.676,155.955
C08469=1052.251,5.650,426.125,170.719,31.677,155.955
C08470=1052.258,5.899,426.110,170.721,31.680,155.956
C08471=1052.264,6.148,426.096,170.723,31.682,155.956
C08472=1052.270,6.398,426.081,170.725,31.684,155.956
C08473=1052.276,6.647,426.065,170.727,31.686,155.956
C08474=1052.282,6.897,426.050,170.728,31.688,155.957
C08475=1052.289,7.146,426.035,170.730,31.690,155.957
C08476=1052.294,7.395,426.020,170.732,31.691,155.957
C08477=1052.301,7.645,426.005,170.734,31.693,155.957
C08478=1052.307,7.895,425.990,170.734,31.695,155.958
C08479=1052.314,8.144,425.974,170.736,31.697,155.958
C08480=1052.320,8.393,425.960,170.738,31.700,155.958
C08481=1052.327,8.643,425.945,170.740,31.702,155.959
C08482=1052.332,8.892,425.929,170.742,31.704,155.959
C08483=1052.338,9.142,425.914,170.743,31.705,155.959
C08484=1052.344,9.392,425.900,170.745,31.707,155.959
C08485=1052.351,9.641,425.884,170.747,31.709,155.960
C08486=1052.358,9.890,425.869,170.749,31.711,155.960
C08487=1052.364,10.140,425.854,170.750,31.713,155.960
C08488=1052.370,10.390,425.839,170.751,31.715,155.961
C08489=1052.377,10.639,425.823,170.753,31.718,155.961
C08490=1052.382,10.888,425.808,170.755,31.719,155.961
C08491=1052.388,11.138,425.793,170.757,31.721,155.961
C08492=1052.395,11.387,425.778,170.758,31.723,155.962
C08493=1052.402,11.636,425.763,170.760,31.725,155.962
C08494=1052.408,11.886,425.748,170.762,31.727,155.962
C08495=1052.414,12.136,425.733,170.764,31.729,155.963
C08496=1052.421,12.385,425.717,170.765,31.731,155.963
C08497=1052.427,12.635,425.702,170.767,31.733,155.963
C08498=1052.433,12.884,425.687,170.768,31.735,155.963
C08499=1052.440,13.169,425.669,170.770,31.737,155.964
C08500=1052.448,13.453,425.653,170.772,31.740,155.964
C08501=1052.455,13.737,425.635,170.774,31.742,155.964
C08502=1052.462,14.022,425.617,170.776,31.744,155.965
C08503=1052.468,14.271,425.602,170.778,31.746,155.965
C08504=1052.474,14.520,425.586,170.779,31.748,155.965
C08505=1052.481,14.770,425.571,170.781,31.750,155.965
C08506=1052.486,15.020,425.556,170.783,31.752,155.966
C08507=1052.493,15.269,425.540,170.784,31.754,155.966
C08508=1052.499,15.519,425.525,170.785,31.756,155.966
C08509=1052.505,15.768,425.509,170.787,31.758,155.967
C08510=1052.512,16.018,425.494,170.789,31.760,155.967
C08511=1052.518,16.267,425.479,170.791,31.762,155.967
C08512=1052.524,16.517,425.463,170.792,31.764,155.968
C08513=1052.530,16.766,425.448,170.794,31.766,155.968
C08514=1052.536,17.016,425.431,170.796,31.769,155.968
C08515=1052.543,17.265,425.416,170.798,31.771,155.968
C08516=1052.549,17.514,425.401,170.799,31.773,155.969
C08517=1052.554,17.764,425.386,170.801,31.775,155.969
C08518=1052.561,18.013,425.370,170.802,31.777,155.969
C08519=1052.567,18.263,425.354,170.804,31.779,155.970
C08520=1052.573,18.512,425.339,170.805,31.781,155.970
C08521=1052.580,18.761,425.324,170.807,31.783,155.970
C08522=1052.586,19.011,425.307,170.809,31.785,155.970
C08523=1052.592,19.260,425.293,170.811,31.787,155.971
C08524=1052.598,19.510,425.276,170.812,31.789,155.971
C08525=1052.605,19.759,425.261,170.814,31.791,155.971
C08526=1052.610,20.009,425.245,170.816,31.793,155.972
C08527=1052.617,20.258,425.229,170.817,31.795,155.972
C08528=1052.623,20.508,425.214,170.818,31.797,155.972
C08529=1052.629,20.757,425.198,170.820,31.799,155.973
C08530=1052.635,21.007,425.183,170.822,31.801,155.973
C08531=1052.642,21.256,425.167,170.823,31.803,155.973
C08532=1052.648,21.505,425.151,170.825,31.805,155.973
C08533=1052.654,21.755,425.136,170.827,31.808,155.974
C08534=1052.660,22.004,425.120,170.829,31.810,155.974
C08535=1052.667,22.253,425.104,170.830,31.812,155.974
C08536=1052.672,22.503,425.088,170.832,31.814,155.975
C08537=1052.679,22.752,425.073,170.834,31.816,155.975
C08538=1052.685,23.002,425.056,170.834,31.818,155.975
C08539=1052.691,23.252,425.041,170.836,31.820,155.976
C08540=1052.697,23.501,425.025,170.838,31.822,155.976
C08541=1052.703,23.750,425.009,170.840,31.825,155.976
C08542=1052.710,24.000,424.994,170.841,31.827,155.977
C08543=1052.716,24.249,424.978,170.843,31.829,155.977
C08544=1052.722,24.498,424.962,170.845,31.831,155.977
C08545=1052.728,24.748,424.947,170.847,31.833,155.977
C08546=1052.734,24.997,424.930,170.848,31.835,155.978
C08547=1052.741,25.246,424.915,170.850,31.837,155.978
C08548=1052.747,25.496,424.898,170.852,31.839,155.978
C08549=1052.754,25.746,424.883,170.852,31.841,155.979
C08550=1052.759,25.995,424.867,170.854,31.843,155.979
C08551=1052.766,26.244,424.851,170.856,31.845,155.979
C08552=1052.772,26.494,424.835,170.858,31.847,155.980
C08553=1052.778,26.744,424.819,170.859,31.849,155.980
C08554=1052.784,26.993,424.804,170.861,31.851,155.980
C08555=1052.790,27.242,424.787,170.863,31.853,155.980
C08556=1052.797,27.491,424.772,170.864,31.855,155.981
C08557=1052.803,27.741,424.756,170.866,31.857,155.981
C08558=1052.809,27.990,424.739,170.868,31.859,155.981
C08559=1052.815,28.240,424.724,170.869,31.862,155.982
C08560=1052.822,28.490,424.708,170.870,31.864,155.982
C08561=1052.828,28.739,424.691,170.872,31.866,155.982
C08562=1052.834,28.988,424.675,170.874,31.868,155.983
C08563=1052.841,29.274,424.657,170.876,31.870,155.983
C08564=1052.848,29.560,424.638,170.878,31.873,155.983
C08565=1052.855,29.846,424.620,170.880,31.876,155.984
C08566=1052.862,30.131,424.602,170.881,31.878,155.984
C08567=1052.868,30.380,424.586,170.883,31.880,155.984
C08568=1052.875,30.630,424.569,170.885,31.882,155.985
C08569=1052.881,30.880,424.553,170.887,31.884,155.985
C08570=1052.887,31.129,424.537,170.887,31.886,155.985
C08571=1052.893,31.378,424.521,170.889,31.888,155.986
C08572=1052.899,31.627,424.505,170.891,31.891,155.986
C08573=1052.905,31.877,424.489,170.892,31.892,155.986
C08574=1052.911,32.126,424.472,170.894,31.895,155.987
C08575=1052.917,32.375,424.456,170.896,31.897,155.987
C08576=1052.924,32.625,424.440,170.897,31.899,155.987
C08577=1052.930,32.874,424.424,170.899,31.901,155.988
C08578=1052.936,33.124,424.408,170.901,31.903,155.988
C08579=1052.942,33.373,424.391,170.903,31.905,155.988
C08580=1052.948,33.622,424.375,170.904,31.907,155.988
C08581=1052.954,33.872,424.359,170.905,31.909,155.989
C08582=1052.962,34.122,424.343,170.907,31.912,155.989
C08583=1052.968,34.371,424.327,170.908,31.914,155.990
C08584=1052.973,34.620,424.310,170.910,31.916,155.990
C08585=1052.979,34.870,424.294,170.912,31.918,155.990
C08586=1052.985,35.119,424.278,170.913,31.920,155.990
C08587=1052.991,35.368,424.262,170.915,31.922,155.991
C08588=1052.999,35.618,424.246,170.917,31.924,155.991
C08589=1053.005,35.867,424.229,170.919,31.926,155.991
C08590=1053.011,36.117,424.213,170.920,31.929,155.992
C08591=1053.016,36.366,424.197,170.922,31.931,155.992
C08592=1053.023,36.616,424.180,170.923,31.933,155.992
C08593=1053.029,36.865,424.164,170.924,31.935,155.993
C08594=1053.036,37.114,424.148,170.926,31.937,155.993
C08595=1053.042,37.363,424.131,170.928,31.939,155.993
C08596=1053.048,37.613,424.115,170.929,31.941,155.994
C08597=1053.054,37.863,424.098,170.931,31.944,155.994
C08598=1053.060,38.112,424.082,170.933,31.946,155.994
C08599=1053.066,38.361,424.066,170.934,31.948,155.995
C08600=1053.073,38.610,424.049,170.936,31.950,155.995
C08601=1053.079,38.860,424.032,170.938,31.953,155.995
C08602=1053.085,39.109,424.016,170.939,31.955,155.996
C08603=1053.091,39.359,424.000,170.940,31.957,155.996
C08604=1053.097,39.608,423.984,170.942,31.959,155.996
C08605=1053.103,39.857,423.967,170.944,31.961,155.996
C08606=1053.110,40.107,423.950,170.945,31.963,155.997
C08607=1053.116,40.356,423.934,170.947,31.965,155.997
C08608=1053.122,40.606,423.917,170.949,31.967,155.997
C08609=1053.127,40.855,423.900,170.950,31.969,155.998
C08610=1053.134,41.105,423.883,170.952,31.972,155.998
C08611=1053.140,41.354,423.867,170.954,31.974,155.998
C08612=1053.146,41.603,423.851,170.955,31.976,155.999
C08613=1053.152,41.852,423.834,170.957,31.978,155.999
C08614=1053.158,42.102,423.817,170.959,31.980,155.999
C08615=1053.164,42.352,423.801,170.959,31.983,156.000
C08616=1053.171,42.600,423.784,170.961,31.985,156.000
C08617=1053.177,42.850,423.768,170.963,31.987,156.000
C08618=1053.183,43.100,423.751,170.964,31.989,156.001
C08619=1053.189,43.348,423.734,170.966,31.992,156.001
C08620=1053.195,43.598,423.718,170.968,31.994,156.001
C08621=1053.201,43.848,423.701,170.969,31.996,156.002
C08622=1053.207,44.097,423.684,170.971,31.998,156.002
C08623=1053.213,44.346,423.667,170.973,32.000,156.002
C08624=1053.220,44.595,423.650,170.974,32.002,156.003
C08625=1053.226,44.845,423.633,170.976,32.005,156.003
C08626=1053.231,45.095,423.617,170.977,32.007,156.003
C08627=1053.238,45.380,423.597,170.979,32.010,156.004
C08628=1053.246,45.665,423.578,170.980,32.012,156.004
C08629=1053.252,45.952,423.559,170.982,32.014,156.005
C08630=1053.259,46.237,423.540,170.984,32.017,156.005
C08631=1053.265,46.487,423.523,170.986,32.020,156.005
C08632=1053.271,46.736,423.506,170.988,32.022,156.006
C08633=1053.277,46.985,423.489,170.989,32.024,156.006
C08634=1053.283,47.235,423.471,170.991,32.026,156.006
C08635=1053.289,47.484,423.455,170.993,32.028,156.007
C08636=1053.296,47.733,423.438,170.994,32.030,156.007
C08637=1053.301,47.983,423.421,170.996,32.033,156.007
C08638=1053.308,48.232,423.404,170.997,32.035,156.008
C08639=1053.314,48.482,423.388,170.998,32.037,156.008
C08640=1053.319,48.731,423.370,171.000,32.039,156.008
C08641=1053.326,48.981,423.354,171.002,32.042,156.009
C08642=1053.332,49.229,423.337,171.003,32.044,156.009
C08643=1053.337,49.479,423.320,171.005,32.046,156.009
C08644=1053.344,49.729,423.302,171.007,32.048,156.010
C08645=1053.350,49.977,423.285,171.008,32.050,156.010
C08646=1053.356,50.227,423.269,171.010,32.052,156.010
C08647=1053.362,50.476,423.251,171.012,32.055,156.011
C08648=1053.368,50.726,423.235,171.013,32.057,156.011
C08649=1053.374,50.975,423.217,171.015,32.059,156.011
C08650=1053.381,51.224,423.200,171.016,32.062,156.012
C08651=1053.387,51.474,423.184,171.017,32.064,156.012
C08652=1053.393,51.723,423.166,171.019,32.066,156.013
C08653=1053.399,51.973,423.150,171.021,32.068,156.013
C08654=1053.405,52.221,423.133,171.022,32.070,156.013
C08655=1053.411,52.471,423.115,171.024,32.072,156.014
C08656=1053.417,52.720,423.098,171.025,32.074,156.014
C08657=1053.424,52.970,423.081,171.027,32.077,156.014
C08658=1053.429,53.219,423.064,171.029,32.079,156.015
C08659=1053.436,53.469,423.047,171.030,32.081,156.015
C08660=1053.442,53.718,423.030,171.032,32.084,156.015
C08661=1053.448,53.967,423.012,171.034,32.086,156.016
C08662=1053.454,54.217,422.996,171.035,32.088,156.016
C08663=1053.460,54.466,422.978,171.036,32.090,156.016
C08664=1053.467,54.715,422.961,171.038,32.092,156.017
C08665=1053.473,54.964,422.944,171.039,32.094,156.017
C08666=1053.479,55.214,422.927,171.041,32.096,156.017
C08667=1053.485,55.463,422.910,171.043,32.099,156.018
C08668=1053.492,55.712,422.892,171.044,32.101,156.018
C08669=1053.497,55.962,422.875,171.046,32.103,156.018
C08670=1053.503,56.211,422.858,171.048,32.106,156.019
C08671=1053.509,56.461,422.841,171.049,32.108,156.019
C08672=1053.516,56.709,422.824,171.051,32.110,156.019
C08673=1053.523,56.959,422.806,171.053,32.112,156.020
C08674=1053.528,57.208,422.789,171.054,32.114,156.020
C08675=1053.535,57.458,422.772,171.056,32.116,156.020
C08676=1053.540,57.707,422.754,171.057,32.118,156.021
C08677=1053.547,57.956,422.737,171.058,32.121,156.021
C08678=1053.553,58.205,422.720,171.060,32.123,156.021
C08679=1053.559,58.455,422.703,171.062,32.125,156.022
C08680=1053.565,58.704,422.686,171.063,32.127,156.022
C08681=1053.571,58.954,422.668,171.065,32.130,156.022
C08682=1053.578,59.203,422.651,171.067,32.132,156.023
C08683=1053.585,59.452,422.634,171.068,32.134,156.023
C08684=1053.591,59.702,422.616,171.070,32.136,156.023
C08685=1053.597,59.951,422.599,171.072,32.138,156.024
C08686=1053.603,60.201,422.582,171.073,32.140,156.024
C08687=1053.609,60.450,422.565,171.075,32.142,156.024
C08688=1053.615,60.699,422.547,171.077,32.145,156.025
C08689=1053.621,60.948,422.530,171.077,32.147,156.025
C08690=1053.628,61.198,422.512,171.079,32.149,156.025
C08691=1053.635,61.483,422.492,171.081,32.152,156.026
C08692=1053.642,61.768,422.472,171.083,32.154,156.026
C08693=1053.650,62.054,422.453,171.085,32.156,156.026
C08694=1053.657,62.340,422.433,171.087,32.159,156.027
C08695=1053.663,62.589,422.415,171.088,32.161,156.027
C08696=1053.669,62.838,422.398,171.090,32.163,156.028
C08697=1053.676,63.087,422.381,171.092,32.166,156.028
C08698=1053.681,63.337,422.363,171.093,32.168,156.028
C08699=1053.688,63.586,422.346,171.095,32.170,156.029
C08700=1053.694,63.836,422.328,171.097,32.172,156.029
C08701=1053.701,64.084,422.311,171.098,32.174,156.029
C08702=1053.707,64.334,422.293,171.099,32.176,156.030
C08703=1053.713,64.583,422.276,171.101,32.178,156.030
C08704=1053.719,64.833,422.258,171.102,32.181,156.030
C08705=1053.725,65.082,422.240,171.104,32.183,156.031
C08706=1053.731,65.331,422.222,171.106,32.185,156.031
C08707=1053.738,65.581,422.205,171.107,32.188,156.031
C08708=1053.743,65.830,422.188,171.109,32.190,156.032
C08709=1053.750,66.079,422.169,171.111,32.192,156.032
C08710=1053.756,66.328,422.152,171.112,32.194,156.032
C08711=1053.762,66.577,422.134,171.114,32.196,156.033
C08712=1053.768,66.827,422.116,171.116,32.199,156.033
C08713=1053.774,67.076,422.099,171.117,32.201,156.033
C08714=1053.780,67.326,422.081,171.119,32.203,156.034
C08715=1053.787,67.575,422.063,171.121,32.206,156.034
C08716=1053.792,67.824,422.046,171.121,32.208,156.034
C08717=1053.799,68.073,422.028,171.123,32.210,156.035
C08718=1053.805,68.322,422.010,171.125,32.212,156.035
C08719=1053.811,68.572,421.992,171.126,32.214,156.035
C08720=1053.817,68.822,421.974,171.128,32.217,156.036
C08721=1053.823,69.071,421.957,171.130,32.219,156.036
C08722=1053.829,69.320,421.939,171.131,32.221,156.037
C08723=1053.836,69.569,421.921,171.133,32.224,156.037
C08724=1053.841,69.818,421.903,171.135,32.226,156.037
C08725=1053.848,70.068,421.886,171.136,32.227,156.038
C08726=1053.854,70.317,421.868,171.138,32.230,156.038
C08727=1053.860,70.566,421.850,171.140,32.232,156.038
C08728=1053.866,70.816,421.832,171.141,32.235,156.039
C08729=1053.872,71.065,421.814,171.143,32.237,156.039
C08730=1053.878,71.315,421.796,171.145,32.239,156.039
C08731=1053.884,71.564,421.777,171.145,32.241,156.040
C08732=1053.890,71.813,421.760,171.147,32.243,156.040
C08733=1053.897,72.062,421.743,171.148,32.246,156.040
C08734=1053.903,72.311,421.724,171.150,32.248,156.041
C08735=1053.909,72.560,421.706,171.152,32.251,156.041
C08736=1053.915,72.810,421.688,171.153,32.253,156.042
C08737=1053.921,73.059,421.670,171.155,32.255,156.042
C08738=1053.927,73.308,421.652,171.157,32.257,156.042
C08739=1053.933,73.558,421.634,171.158,32.259,156.043
C08740=1053.939,73.807,421.616,171.160,32.262,156.043
C08741=1053.945,74.056,421.598,171.162,32.264,156.043
C08742=1053.951,74.306,421.580,171.163,32.266,156.044
C08743=1053.957,74.555,421.561,171.165,32.268,156.044
C08744=1053.964,74.804,421.544,171.167,32.271,156.044
C08745=1053.970,75.053,421.527,171.168,32.273,156.045
C08746=1053.976,75.303,421.508,171.169,32.275,156.045
C08747=1053.982,75.552,421.490,171.171,32.278,156.045
C08748=1053.988,75.801,421.472,171.172,32.280,156.046
C08749=1053.994,76.050,421.454,171.174,32.282,156.046
C08750=1054.000,76.300,421.436,171.176,32.284,156.047
C08751=1054.006,76.549,421.418,171.177,32.286,156.047
C08752=1054.012,76.798,421.400,171.179,32.289,156.047
C08753=1054.019,77.047,421.381,171.181,32.291,156.048
C08754=1054.025,77.297,421.363,171.182,32.293,156.048
C08755=1054.032,77.583,421.342,171.184,32.296,156.048
C08756=1054.039,77.867,421.322,171.186,32.298,156.049
C08757=1054.045,78.153,421.301,171.188,32.301,156.049
C08758=1054.052,78.438,421.280,171.190,32.303,156.050
C08759=1054.058,78.681,421.262,171.191,32.305,156.050
C08760=1054.065,78.925,421.244,171.193,32.308,156.050
C08761=1054.071,79.168,421.226,171.194,32.310,156.051
C08762=1054.076,79.411,421.209,171.195,32.313,156.051
C08763=1054.082,79.654,421.191,171.197,32.315,156.051
C08764=1054.088,79.897,421.173,171.199,32.317,156.052
C08765=1054.093,80.140,421.155,171.200,32.319,156.052
C08766=1054.099,80.383,421.137,171.202,32.321,156.052
C08767=1054.105,80.633,421.118,171.203,32.324,156.053
C08768=1054.112,80.882,421.100,171.205,32.326,156.053
C08769=1054.118,81.131,421.082,171.207,32.328,156.054
C08770=1054.124,81.380,421.063,171.208,32.330,156.054
C08771=1054.130,81.629,421.045,171.210,32.333,156.054
C08772=1054.136,81.879,421.026,171.212,32.335,156.055
C08773=1054.142,82.128,421.008,171.213,32.338,156.055
C08774=1054.148,82.377,420.990,171.215,32.340,156.055
C08775=1054.154,82.626,420.971,171.217,32.342,156.056
C08776=1054.160,82.875,420.953,171.218,32.344,156.056
C08777=1054.166,83.126,420.934,171.219,32.347,156.056
C08778=1054.172,83.375,420.916,171.221,32.349,156.057
C08779=1054.178,83.623,420.897,171.222,32.351,156.057
C08780=1054.184,83.873,420.879,171.224,32.353,156.058
C08781=1054.191,84.122,420.861,171.226,32.356,156.058
C08782=1054.196,84.371,420.841,171.227,32.358,156.058
C08783=1054.203,84.620,420.823,171.229,32.361,156.059
C08784=1054.208,84.869,420.805,171.231,32.363,156.059
C08785=1054.215,85.119,420.787,171.232,32.365,156.059
C08786=1054.221,85.368,420.768,171.234,32.367,156.060
C08787=1054.227,85.617,420.749,171.236,32.369,156.060
C08788=1054.233,85.867,420.731,171.237,32.372,156.060
C08789=1054.239,86.116,420.712,171.239,32.374,156.061
C08790=1054.246,86.365,420.693,171.241,32.377,156.061
C08791=1054.251,86.614,420.675,171.242,32.378,156.061
C08792=1054.257,86.864,420.657,171.244,32.381,156.062
C08793=1054.263,87.113,420.638,171.246,32.383,156.062
C08794=1054.270,87.362,420.619,171.246,32.386,156.063
C08795=1054.275,87.611,420.600,171.248,32.388,156.063
C08796=1054.282,87.860,420.581,171.250,32.390,156.063
C08797=1054.288,88.110,420.564,171.251,32.392,156.064
C08798=1054.294,88.359,420.545,171.253,32.394,156.064
C08799=1054.300,88.608,420.527,171.255,32.397,156.064
C08800=1054.306,88.857,420.507,171.256,32.399,156.065
C08801=1054.312,89.106,420.489,171.258,32.401,156.065
C08802=1054.319,89.355,420.470,171.260,32.403,156.065
C08803=1054.325,89.605,420.451,171.261,32.406,156.066
C08804=1054.331,89.855,420.433,171.263,32.408,156.066
C08805=1054.337,90.104,420.414,171.265,32.410,156.067
C08806=1054.343,90.353,420.396,171.266,32.413,156.067
C08807=1054.349,90.602,420.376,171.268,32.415,156.067
C08808=1054.356,90.851,420.358,171.270,32.417,156.068
C08809=1054.361,91.101,420.338,171.271,32.419,156.068
C08810=1054.368,91.350,420.320,171.273,32.422,156.068
C08811=1054.373,91.599,420.301,171.275,32.424,156.069
C08812=1054.379,91.848,420.282,171.275,32.426,156.069
C08813=1054.386,92.097,420.264,171.277,32.429,156.070
C08814=1054.391,92.346,420.244,171.279,32.431,156.070
C08815=1054.398,92.595,420.226,171.280,32.434,156.070
C08816=1054.403,92.845,420.207,171.282,32.436,156.071
C08817=1054.410,93.094,420.188,171.284,32.438,156.071
C08818=1054.416,93.343,420.169,171.285,32.440,156.071
C08819=1054.423,93.640,420.146,171.287,32.443,156.072
C08820=1054.429,93.938,420.124,171.289,32.446,156.072
C08821=1054.437,94.236,420.101,171.291,32.449,156.073
C08822=1054.444,94.533,420.078,171.293,32.451,156.073
C08823=1054.450,94.782,420.059,171.295,32.454,156.074
C08824=1054.456,95.032,420.040,171.297,32.456,156.074
C08825=1054.462,95.281,420.021,171.298,32.458,156.074
C08826=1054.469,95.530,420.003,171.300,32.460,156.075
C08827=1054.474,95.780,419.983,171.302,32.463,156.075
C08828=1054.481,96.029,419.965,171.303,32.465,156.075
C08829=1054.486,96.278,419.945,171.305,32.468,156.076
C08830=1054.492,96.528,419.926,171.306,32.470,156.076
C08831=1054.499,96.776,419.907,171.307,32.472,156.077
C08832=1054.504,97.025,419.888,171.309,32.474,156.077
C08833=1054.511,97.275,419.869,171.311,32.477,156.077
C08834=1054.517,97.524,419.850,171.313,32.479,156.078
C08835=1054.523,97.773,419.831,171.314,32.481,156.078
C08836=1054.529,98.023,419.812,171.316,32.483,156.078
C08837=1054.535,98.271,419.792,171.318,32.486,156.079
C08838=1054.541,98.520,419.773,171.319,32.488,156.079
C08839=1054.548,98.770,419.755,171.321,32.491,156.080
C08840=1054.553,99.019,419.735,171.323,32.493,156.080
C08841=1054.560,99.268,419.717,171.324,32.495,156.080
C08842=1054.566,99.517,419.697,171.326,32.497,156.081
C08843=1054.571,99.766,419.677,171.328,32.500,156.081
C08844=1054.578,100.016,419.659,171.329,32.502,156.081
C08845=1054.583,100.265,419.640,171.331,32.504,156.082
C08846=1054.590,100.514,419.621,171.333,32.506,156.082
C08847=1054.596,100.763,419.601,171.335,32.509,156.082
C08848=1054.602,101.012,419.582,171.336,32.511,156.083
C08849=1054.608,101.261,419.563,171.338,32.514,156.083
C08850=1054.614,101.510,419.543,171.340,32.516,156.084
C08851=1054.620,101.760,419.524,171.340,32.518,156.084
C08852=1054.626,102.010,419.504,171.342,32.521,156.084
C08853=1054.633,102.258,419.485,171.344,32.523,156.085
C08854=1054.638,102.508,419.466,171.345,32.525,156.085
C08855=1054.644,102.757,419.446,171.347,32.528,156.086
C08856=1054.650,103.006,419.426,171.349,32.530,156.086
C08857=1054.656,103.255,419.407,171.350,32.532,156.086
C08858=1054.662,103.505,419.389,171.352,32.535,156.087
C08859=1054.668,103.753,419.369,171.354,32.537,156.087
C08860=1054.674,104.003,419.349,171.355,32.540,156.087
C08861=1054.680,104.252,419.330,171.357,32.542,156.088
C08862=1054.686,104.501,419.310,171.359,32.544,156.088
C08863=1054.692,104.750,419.292,171.361,32.546,156.088
C08864=1054.698,104.999,419.272,171.362,32.549,156.089
C08865=1054.704,105.248,419.252,171.364,32.551,156.089
C08866=1054.710,105.497,419.232,171.366,32.553,156.090
C08867=1054.715,105.747,419.213,171.367,32.556,156.090
C08868=1054.722,105.997,419.193,171.369,32.558,156.090
C08869=1054.728,106.245,419.174,171.371,32.561,156.091
C08870=1054.734,106.495,419.155,171.372,32.562,156.091
C08871=1054.740,106.744,419.135,171.374,32.565,156.092
C08872=1054.746,106.993,419.116,171.375,32.568,156.092
C08873=1054.752,107.242,419.096,171.377,32.570,156.092
C08874=1054.758,107.491,419.077,171.378,32.572,156.093
C08875=1054.764,107.740,419.057,171.380,32.574,156.093
C08876=1054.770,107.990,419.038,171.382,32.577,156.093
C08877=1054.776,108.239,419.018,171.383,32.579,156.094
C08878=1054.782,108.488,418.998,171.385,32.581,156.094
C08879=1054.788,108.737,418.978,171.387,32.584,156.095
C08880=1054.794,108.986,418.958,171.389,32.586,156.095
C08881=1054.801,109.235,418.940,171.390,32.589,156.095
C08882=1054.807,109.484,418.920,171.392,32.591,156.096
C08883=1054.813,109.770,418.897,171.394,32.593,156.096
C08884=1054.820,110.055,418.875,171.396,32.596,156.097
C08885=1054.827,110.340,418.853,171.398,32.598,156.097
C08886=1054.835,110.625,418.830,171.400,32.601,156.097
C08887=1054.841,110.875,418.810,171.402,32.604,156.098
C08888=1054.847,111.124,418.790,171.403,32.606,156.098
C08889=1054.853,111.373,418.771,171.405,32.608,156.099
C08890=1054.859,111.622,418.751,171.407,32.611,156.099
C08891=1054.865,111.871,418.731,171.408,32.613,156.099
C08892=1054.870,112.120,418.712,171.410,32.615,156.100
C08893=1054.877,112.370,418.692,171.412,32.618,156.100
C08894=1054.883,112.619,418.672,171.414,32.620,156.100
C08895=1054.889,112.868,418.652,171.415,32.622,156.101
C08896=1054.895,113.117,418.632,171.416,32.624,156.101
C08897=1054.901,113.366,418.612,171.418,32.627,156.102
C08898=1054.907,113.615,418.592,171.419,32.630,156.102
C08899=1054.913,113.865,418.573,171.421,32.632,156.102
C08900=1054.919,114.113,418.553,171.423,32.634,156.103
C08901=1054.924,114.362,418.532,171.425,32.637,156.103
C08902=1054.930,114.611,418.512,171.426,32.639,156.104
C08903=1054.936,114.861,418.493,171.428,32.641,156.104
C08904=1054.942,115.110,418.473,171.430,32.644,156.104
C08905=1054.948,115.359,418.453,171.431,32.646,156.105
C08906=1054.954,115.608,418.432,171.433,32.649,156.105
C08907=1054.960,115.857,418.412,171.435,32.651,156.106
C08908=1054.965,116.106,418.393,171.437,32.654,156.106
C08909=1054.972,116.356,418.373,171.438,32.656,156.106
C08910=1054.977,116.605,418.352,171.440,32.658,156.107
C08911=1054.983,116.854,418.332,171.442,32.661,156.107
C08912=1054.989,117.103,418.312,171.444,32.663,156.108
C08913=1054.995,117.351,418.292,171.445,32.665,156.108
C08914=1055.001,117.601,418.271,171.447,32.668,156.108
C08915=1055.007,117.850,418.251,171.449,32.671,156.109
C08916=1055.013,118.100,418.232,171.450,32.673,156.109
C08917=1055.019,118.348,418.212,171.452,32.675,156.110
C08918=1055.025,118.598,418.191,171.454,32.678,156.110
C08919=1055.031,118.847,418.171,171.456,32.680,156.110
C08920=1055.036,119.096,418.151,171.457,32.682,156.111
C08921=1055.042,119.345,418.131,171.459,32.685,156.111
C08922=1055.048,119.594,418.111,171.461,32.687,156.111
C08923=1055.054,119.843,418.091,171.462,32.689,156.112
C08924=1055.060,120.092,418.071,171.463,32.692,156.112
C08925=1055.066,120.341,418.050,171.465,32.694,156.113
C08926=1055.072,120.591,418.030,171.467,32.697,156.113
C08927=1055.078,120.840,418.010,171.469,32.699,156.114
C08928=1055.084,121.088,417.990,171.470,32.701,156.114
C08929=1055.090,121.338,417.969,171.472,32.704,156.114
C08930=1055.096,121.587,417.949,171.474,32.706,156.115
C08931=1055.102,121.836,417.929,171.476,32.708,156.115
C08932=1055.108,122.086,417.908,171.477,32.711,156.115
C08933=1055.114,122.334,417.888,171.479,32.713,156.116
C08934=1055.120,122.583,417.868,171.481,32.716,156.116
C08935=1055.126,122.833,417.847,171.483,32.718,156.117
C08936=1055.132,123.082,417.827,171.484,32.721,156.117
C08937=1055.138,123.331,417.807,171.486,32.723,156.117
C08938=1055.144,123.580,417.787,171.488,32.725,156.118
C08939=1055.150,123.829,417.766,171.490,32.728,156.118
C08940=1055.156,124.078,417.746,171.491,32.730,156.119
C08941=1055.162,124.327,417.725,171.493,32.732,156.119
C08942=1055.168,124.576,417.705,171.495,32.735,156.119
C08943=1055.174,124.825,417.685,171.497,32.737,156.120
C08944=1055.180,125.075,417.665,171.498,32.739,156.120
C08945=1055.186,125.324,417.644,171.500,32.742,156.121
C08946=1055.192,125.572,417.624,171.502,32.744,156.121
C08947=1055.199,125.858,417.600,171.504,32.747,156.121
C08948=1055.206,126.143,417.577,171.506,32.750,156.122
C08949=1055.212,126.428,417.553,171.508,32.752,156.122
C08950=1055.220,126.713,417.530,171.510,32.755,156.123
C08951=1055.226,126.963,417.510,171.512,32.758,156.123
C08952=1055.232,127.212,417.490,171.514,32.760,156.123
C08953=1055.238,127.460,417.470,171.515,32.762,156.124
C08954=1055.244,127.710,417.448,171.516,32.765,156.124
C08955=1055.250,127.958,417.428,171.518,32.767,156.125
C08956=1055.256,128.208,417.408,171.520,32.769,156.125
C08957=1055.262,128.457,417.387,171.522,32.771,156.125
C08958=1055.268,128.706,417.366,171.523,32.774,156.126
C08959=1055.274,128.955,417.346,171.525,32.776,156.126
C08960=1055.280,129.205,417.325,171.527,32.778,156.127
C08961=1055.286,129.453,417.305,171.529,32.781,156.127
C08962=1055.292,129.702,417.284,171.531,32.784,156.127
C08963=1055.298,129.951,417.264,171.532,32.786,156.128
C08964=1055.304,130.200,417.244,171.534,32.788,156.128
C08965=1055.311,130.449,417.222,171.536,32.790,156.129
C08966=1055.317,130.698,417.202,171.538,32.793,156.129
C08967=1055.323,130.948,417.182,171.540,32.795,156.129
C08968=1055.329,131.196,417.160,171.541,32.797,156.130
C08969=1055.335,131.446,417.140,171.543,32.800,156.130
C08970=1055.341,131.695,417.120,171.545,32.802,156.131
C08971=1055.348,131.944,417.099,171.547,32.804,156.131
C08972=1055.353,132.193,417.078,171.549,32.807,156.131
C08973=1055.359,132.442,417.058,171.550,32.810,156.132
C08974=1055.365,132.691,417.036,171.552,32.812,156.132
C08975=1055.371,132.941,417.016,171.554,32.814,156.132
C08976=1055.377,133.189,416.995,171.556,32.817,156.133
C08977=1055.383,133.439,416.974,171.558,32.819,156.133
C08978=1055.389,133.687,416.953,171.559,32.822,156.134
C08979=1055.395,133.936,416.933,171.561,32.824,156.134
C08980=1055.401,134.185,416.911,171.563,32.826,156.135
C08981=1055.406,134.434,416.890,171.565,32.829,156.135
C08982=1055.413,134.683,416.869,171.567,32.832,156.135
C08983=1055.418,134.932,416.849,171.568,32.833,156.136
C08984=1055.424,135.182,416.827,171.570,32.836,156.136
C08985=1055.430,135.431,416.807,171.572,32.839,156.137
C08986=1055.436,135.680,416.786,171.574,32.841,156.137
C08987=1055.442,135.929,416.765,171.576,32.843,156.137
C08988=1055.449,136.178,416.744,171.577,32.846,156.138
C08989=1055.454,136.428,416.723,171.579,32.848,156.138
C08990=1055.460,136.676,416.702,171.581,32.851,156.139
C08991=1055.467,136.926,416.682,171.583,32.853,156.139
C08992=1055.472,137.174,416.660,171.584,32.856,156.139
C08993=1055.478,137.423,416.639,171.586,32.858,156.140
C08994=1055.484,137.672,416.619,171.587,32.860,156.140
C08995=1055.490,137.921,416.597,171.589,32.863,156.141
C08996=1055.496,138.170,416.577,171.591,32.865,156.141
C08997=1055.502,138.420,416.555,171.593,32.868,156.141
C08998=1055.508,138.668,416.534,171.595,32.870,156.142
C08999=1055.514,138.918,416.513,171.597,32.872,156.142
C09000=1055.520,139.167,416.492,171.598,32.875,156.143
C09001=1055.526,139.415,416.470,171.600,32.877,156.143
C09002=1055.532,139.665,416.450,171.602,32.880,156.143
C09003=1055.538,139.913,416.429,171.604,32.882,156.144
C09004=1055.544,140.163,416.407,171.606,32.885,156.144
C09005=1055.549,140.412,416.387,171.608,32.887,156.145
C09006=1055.555,140.661,416.365,171.609,32.890,156.145
C09007=1055.561,140.909,416.344,171.611,32.892,156.146
C09008=1055.567,141.159,416.322,171.613,32.894,156.146
C09009=1055.574,141.408,416.302,171.615,32.897,156.146
C09010=1055.579,141.657,416.280,171.617,32.899,156.147
C09011=1055.586,141.942,416.255,171.619,32.902,156.147
C09012=1055.593,142.227,416.232,171.621,32.905,156.148
C09013=1055.600,142.512,416.207,171.623,32.908,156.148
C09014=1055.607,142.797,416.183,171.625,32.911,156.149
C09015=1055.612,143.045,416.161,171.627,32.913,156.149
C09016=1055.618,143.295,416.140,171.629,32.916,156.149
C09017=1055.624,143.544,416.119,171.631,32.918,156.150
C09018=1055.630,143.793,416.097,171.633,32.921,156.150
C09019=1055.636,144.042,416.076,171.634,32.923,156.151
C09020=1055.642,144.291,416.055,171.636,32.926,156.151
C09021=1055.648,144.540,416.033,171.638,32.928,156.151
C09022=1055.654,144.789,416.011,171.640,32.930,156.152
C09023=1055.660,145.038,415.991,171.642,32.933,156.152
C09024=1055.666,145.287,415.970,171.644,32.936,156.153
C09025=1055.672,145.536,415.948,171.646,32.938,156.153
C09026=1055.678,145.785,415.927,171.648,32.940,156.154
C09027=1055.684,146.034,415.905,171.649,32.943,156.154
C09028=1055.690,146.283,415.883,171.651,32.945,156.154
C09029=1055.696,146.532,415.862,171.653,32.948,156.155
C09030=1055.702,146.781,415.841,171.655,32.950,156.155
C09031=1055.708,147.030,415.819,171.657,32.952,156.156
C09032=1055.714,147.279,415.798,171.659,32.955,156.156
C09033=1055.720,147.528,415.776,171.661,32.958,156.156
C09034=1055.726,147.777,415.754,171.663,32.960,156.157
C09035=1055.732,148.026,415.733,171.664,32.963,156.157
C09036=1055.738,148.275,415.711,171.666,32.965,156.158
C09037=1055.744,148.524,415.690,171.668,32.967,156.158
C09038=1055.750,148.773,415.668,171.670,32.970,156.158
C09039=1055.756,149.022,415.647,171.672,32.972,156.159
C09040=1055.761,149.271,415.625,171.674,32.975,156.159
C09041=1055.767,149.520,415.603,171.676,32.978,156.160
C09042=1055.773,149.769,415.582,171.678,32.980,156.160
C09043=1055.779,150.018,415.560,171.679,32.983,156.161
C09044=1055.785,150.267,415.539,171.681,32.985,156.161
C09045=1055.791,150.516,415.517,171.683,32.988,156.162
C09046=1055.797,150.765,415.496,171.685,32.990,156.162
C09047=1055.803,151.014,415.473,171.687,32.992,156.162
C09048=1055.809,151.263,415.451,171.689,32.995,156.163
C09049=1055.814,151.512,415.430,171.691,32.997,156.163
C09050=1055.820,151.761,415.408,171.693,33.000,156.164
C09051=1055.827,152.010,415.387,171.695,33.003,156.164
C09052=1055.833,152.259,415.365,171.697,33.005,156.164
C09053=1055.838,152.508,415.343,171.698,33.008,156.165
C09054=1055.844,152.757,415.321,171.700,33.010,156.165
C09055=1055.850,153.006,415.299,171.702,33.013,156.166
C09056=1055.856,153.255,415.277,171.704,33.015,156.166
C09057=1055.862,153.504,415.256,171.705,33.017,156.167
C09058=1055.867,153.753,415.234,171.707,33.020,156.167
C09059=1055.874,154.002,415.212,171.709,33.023,156.167
C09060=1055.880,154.251,415.190,171.711,33.025,156.168
C09061=1055.886,154.499,415.169,171.713,33.028,156.168
C09062=1055.892,154.749,415.147,171.715,33.030,156.169
C09063=1055.897,154.998,415.124,171.717,33.033,156.169
C09064=1055.904,155.247,415.102,171.719,33.035,156.170
C09065=1055.910,155.496,415.081,171.720,33.038,156.170
C09066=1055.915,155.744,415.058,171.722,33.041,156.170
C09067=1055.921,155.993,415.037,171.724,33.043,156.171
C09068=1055.927,156.243,415.015,171.726,33.045,156.171
C09069=1055.933,156.491,414.992,171.728,33.048,156.172
C09070=1055.939,156.741,414.970,171.730,33.050,156.172
C09071=1055.945,156.989,414.949,171.732,33.053,156.173
C09072=1055.950,157.238,414.926,171.734,33.055,156.173
C09073=1055.957,157.487,414.904,171.736,33.058,156.173
C09074=1055.963,157.736,414.883,171.738,33.061,156.174
C09075=1055.970,158.021,414.857,171.740,33.064,156.174
C09076=1055.976,158.306,414.832,171.742,33.066,156.175
C09077=1055.983,158.590,414.807,171.745,33.070,156.175
C09078=1055.990,158.876,414.782,171.747,33.072,156.176
C09079=1055.996,159.124,414.759,171.749,33.075,156.176
C09080=1056.002,159.374,414.737,171.751,33.077,156.177
C09081=1056.007,159.621,414.715,171.753,33.080,156.177
C09082=1056.014,159.871,414.693,171.755,33.082,156.178
C09083=1056.019,160.120,414.670,171.757,33.085,156.178
C09084=1056.026,160.369,414.649,171.758,33.087,156.178
C09085=1056.031,160.618,414.626,171.760,33.090,156.179
C09086=1056.037,160.867,414.604,171.762,33.093,156.179
C09087=1056.043,161.116,414.581,171.764,33.095,156.180
C09088=1056.049,161.364,414.560,171.766,33.098,156.180
C09089=1056.054,161.613,414.537,171.768,33.100,156.181
C09090=1056.060,161.862,414.514,171.770,33.103,156.181
C09091=1056.066,162.111,414.492,171.772,33.106,156.182
C09092=1056.072,162.360,414.470,171.774,33.109,156.182
C09093=1056.077,162.610,414.447,171.776,33.111,156.182
C09094=1056.083,162.858,414.425,171.778,33.114,156.183
C09095=1056.089,163.106,414.402,171.780,33.116,156.183
C09096=1056.095,163.356,414.380,171.782,33.119,156.184
C09097=1056.100,163.605,414.357,171.784,33.122,156.184
C09098=1056.106,163.854,414.334,171.786,33.125,156.185
C09099=1056.112,164.103,414.313,171.788,33.127,156.185
C09100=1056.118,164.352,414.290,171.790,33.130,156.186
C09101=1056.123,164.600,414.267,171.792,33.132,156.186
C09102=1056.128,164.850,414.245,171.794,33.135,156.186
C09103=1056.135,165.098,414.222,171.796,33.137,156.187
C09104=1056.141,165.347,414.200,171.798,33.141,156.187
C09105=1056.146,165.596,414.177,171.800,33.143,156.188
C09106=1056.152,165.846,414.154,171.802,33.146,156.188
